C09062=1058.680,384.878,-115.207,174.460,37.992,157.227
C09063=1058.673,384.632,-115.166,174.454,37.986,157.226
C09064=1058.665,384.385,-115.126,174.449,37.979,157.224
C09065=1058.657,384.139,-115.086,174.443,37.972,157.222
C09066=1058.650,383.892,-115.045,174.437,37.965,157.221
C09067=1058.642,383.646,-115.004,174.432,37.959,157.219
C09068=1058.635,383.399,-114.964,174.427,37.952,157.217
C09069=1058.627,383.153,-114.923,174.420,37.945,157.215
C09070=1058.619,382.906,-114.883,174.415,37.939,157.214
C09071=1058.612,382.659,-114.842,174.409,37.932,157.212
C09072=1058.605,382.414,-114.802,174.404,37.926,157.210
C09073=1058.597,382.167,-114.762,174.399,37.919,157.209
C09074=1058.590,381.920,-114.720,174.392,37.912,157.207
C09075=1058.582,381.673,-114.681,174.387,37.906,157.205
C09076=1058.575,381.428,-114.640,174.382,37.899,157.204
C09077=1058.568,381.180,-114.600,174.377,37.893,157.202
C09078=1058.560,380.933,-114.560,174.371,37.886,157.200
C09079=1058.552,380.687,-114.519,174.366,37.880,157.199
C09080=1058.545,380.441,-114.479,174.360,37.873,157.197
C09081=1058.538,380.194,-114.439,174.354,37.867,157.195
C09082=1058.530,379.947,-114.399,174.349,37.860,157.194
C09083=1058.522,379.701,-114.359,174.344,37.854,157.192
C09084=1058.515,379.454,-114.319,174.339,37.848,157.191
C09085=1058.507,379.207,-114.279,174.333,37.841,157.189
C09086=1058.499,378.961,-114.239,174.327,37.835,157.187
C09087=1058.492,378.714,-114.200,174.322,37.829,157.186
C09088=1058.485,378.467,-114.160,174.317,37.822,157.184
C09089=1058.477,378.221,-114.120,174.311,37.816,157.183
C09090=1058.470,377.974,-114.080,174.306,37.810,157.181
C09091=1058.462,377.727,-114.040,174.301,37.803,157.179
C09092=1058.454,377.481,-114.000,174.296,37.797,157.178
C09093=1058.447,377.234,-113.961,174.291,37.791,157.176
C09094=1058.439,376.987,-113.921,174.285,37.785,157.175
C09095=1058.432,376.741,-113.881,174.280,37.778,157.173
C09096=1058.425,376.494,-113.841,174.274,37.772,157.172
C09097=1058.417,376.248,-113.802,174.269,37.766,157.170
C09098=1058.410,376.001,-113.762,174.264,37.760,157.168
C09099=1058.402,375.754,-113.723,174.258,37.753,157.167
C09100=1058.395,375.508,-113.683,174.253,37.747,157.165
C09101=1058.388,375.261,-113.644,174.248,37.741,157.164
C09102=1058.380,375.014,-113.604,174.243,37.735,157.162
C09103=1058.374,374.768,-113.565,174.238,37.729,157.161
C09104=1058.366,374.521,-113.525,174.232,37.723,157.159
C09105=1058.359,374.274,-113.485,174.227,37.717,157.158
C09106=1058.350,373.998,-113.441,174.222,37.709,157.156
C09107=1058.342,373.723,-113.397,174.216,37.703,157.154
C09108=1058.334,373.447,-113.353,174.210,37.696,157.152
C09109=1058.326,373.172,-113.309,174.204,37.689,157.151
C09110=1058.319,372.924,-113.270,174.199,37.683,157.149
C09111=1058.312,372.678,-113.231,174.194,37.677,157.148
C09112=1058.305,372.431,-113.192,174.189,37.671,157.146
C09113=1058.297,372.184,-113.152,174.184,37.665,157.145
C09114=1058.290,371.938,-113.114,174.179,37.659,157.143
C09115=1058.282,371.690,-113.074,174.174,37.653,157.142
C09116=1058.275,371.444,-113.035,174.169,37.647,157.140
C09117=1058.268,371.197,-112.997,174.164,37.641,157.139
C09118=1058.260,370.950,-112.957,174.159,37.635,157.137
C09119=1058.252,370.704,-112.918,174.154,37.630,157.136
C09120=1058.245,370.457,-112.880,174.149,37.624,157.134
C09121=1058.238,370.210,-112.840,174.144,37.618,157.133
C09122=1058.231,369.963,-112.802,174.139,37.612,157.131
C09123=1058.224,369.716,-112.763,174.134,37.606,157.130
C09124=1058.216,369.469,-112.723,174.128,37.600,157.129
C09125=1058.208,369.223,-112.685,174.123,37.594,157.127
C09126=1058.202,368.976,-112.646,174.118,37.588,157.126
C09127=1058.194,368.729,-112.607,174.113,37.582,157.124
C09128=1058.187,368.482,-112.569,174.109,37.577,157.123
C09129=1058.180,368.235,-112.530,174.104,37.571,157.121
C09130=1058.172,367.989,-112.492,174.099,37.565,157.120
C09131=1058.166,367.742,-112.453,174.094,37.559,157.119
C09132=1058.158,367.494,-112.414,174.089,37.554,157.117
C09133=1058.151,367.248,-112.375,174.084,37.548,157.116
C09134=1058.144,367.001,-112.337,174.079,37.542,157.114
C09135=1058.136,366.754,-112.298,174.075,37.536,157.113
C09136=1058.130,366.507,-112.260,174.070,37.531,157.112
C09137=1058.122,366.261,-112.222,174.065,37.525,157.110
C09138=1058.115,366.013,-112.183,174.060,37.519,157.109
C09139=1058.108,365.766,-112.144,174.055,37.514,157.107
C09140=1058.100,365.520,-112.106,174.051,37.508,157.106
C09141=1058.094,365.272,-112.068,174.046,37.502,157.105
C09142=1058.086,365.026,-112.029,174.041,37.497,157.103
C09143=1058.079,364.779,-111.991,174.036,37.491,157.102
C09144=1058.072,364.532,-111.952,174.031,37.485,157.100
C09145=1058.065,364.285,-111.914,174.027,37.480,157.099
C09146=1058.059,364.038,-111.875,174.022,37.474,157.098
C09147=1058.051,363.791,-111.838,174.017,37.469,157.096
C09148=1058.044,363.544,-111.800,174.012,37.462,157.095
C09149=1058.037,363.298,-111.761,174.007,37.457,157.093
C09150=1058.030,363.050,-111.723,174.003,37.451,157.092
C09151=1058.022,362.804,-111.685,173.998,37.446,157.091
C09152=1058.016,362.557,-111.647,173.993,37.440,157.089
C09153=1058.008,362.309,-111.609,173.988,37.435,157.088
C09154=1058.001,362.063,-111.571,173.984,37.429,157.087
C09155=1057.994,361.815,-111.533,173.979,37.424,157.085
C09156=1057.987,361.569,-111.495,173.974,37.419,157.084
C09157=1057.980,361.322,-111.457,173.969,37.413,157.083
C09158=1057.973,361.074,-111.419,173.965,37.408,157.081
C09159=1057.966,360.828,-111.381,173.960,37.402,157.080
C09160=1057.958,360.581,-111.343,173.955,37.397,157.079
C09161=1057.951,360.334,-111.306,173.951,37.391,157.077
C09162=1057.944,360.076,-111.266,173.946,37.386,157.076
C09163=1057.937,359.819,-111.227,173.941,37.380,157.075
C09164=1057.929,359.562,-111.187,173.936,37.375,157.073
C09165=1057.922,359.304,-111.148,173.931,37.369,157.072
C09166=1057.914,359.057,-111.111,173.926,37.364,157.071
C09167=1057.907,358.810,-111.073,173.922,37.358,157.069
C09168=1057.901,358.563,-111.035,173.917,37.353,157.068
C09169=1057.893,358.315,-110.997,173.912,37.347,157.067
C09170=1057.887,358.069,-110.960,173.908,37.342,157.066
C09171=1057.880,357.822,-110.923,173.904,37.337,157.064
C09172=1057.872,357.575,-110.885,173.899,37.331,157.063
C09173=1057.865,357.328,-110.848,173.895,37.326,157.062
C09174=1057.858,357.080,-110.810,173.890,37.321,157.060
C09175=1057.851,356.833,-110.773,173.886,37.316,157.059
C09176=1057.843,356.586,-110.735,173.881,37.310,157.058
C09177=1057.837,356.340,-110.698,173.876,37.305,157.057
C09178=1057.829,356.093,-110.660,173.872,37.300,157.055
C09179=1057.823,355.845,-110.622,173.867,37.295,157.054
C09180=1057.816,355.597,-110.585,173.862,37.289,157.053
C09181=1057.809,355.350,-110.548,173.859,37.284,157.052
C09182=1057.802,355.104,-110.511,173.854,37.279,157.050
C09183=1057.795,354.857,-110.473,173.850,37.274,157.049
C09184=1057.788,354.610,-110.436,173.845,37.269,157.048
C09185=1057.781,354.363,-110.399,173.840,37.264,157.047
C09186=1057.774,354.115,-110.362,173.836,37.258,157.045
C09187=1057.767,353.868,-110.324,173.831,37.253,157.044
C09188=1057.760,353.621,-110.287,173.827,37.248,157.043
C09189=1057.753,353.374,-110.250,173.823,37.243,157.042
C09190=1057.746,353.126,-110.213,173.818,37.238,157.040
C09191=1057.739,352.879,-110.176,173.814,37.232,157.039
C09192=1057.732,352.633,-110.139,173.809,37.227,157.038
C09193=1057.725,352.385,-110.102,173.805,37.222,157.037
C09194=1057.718,352.139,-110.065,173.800,37.217,157.035
C09195=1057.711,351.891,-110.029,173.796,37.212,157.034
C09196=1057.704,351.644,-109.991,173.792,37.207,157.033
C09197=1057.698,351.397,-109.955,173.788,37.202,157.032
C09198=1057.690,351.150,-109.917,173.783,37.197,157.031
C09199=1057.683,350.902,-109.880,173.779,37.192,157.029
C09200=1057.677,350.655,-109.844,173.774,37.187,157.028
C09201=1057.669,350.408,-109.807,173.770,37.182,157.027
C09202=1057.659,350.018,-109.749,173.763,37.174,157.025
C09203=1057.647,349.628,-109.691,173.756,37.166,157.023
C09204=1057.637,349.238,-109.633,173.750,37.158,157.021
C09205=1057.625,348.847,-109.576,173.742,37.151,157.020
C09206=1057.619,348.601,-109.539,173.739,37.145,157.018
C09207=1057.612,348.353,-109.502,173.734,37.140,157.017
C09208=1057.605,348.106,-109.466,173.730,37.135,157.016
C09209=1057.598,347.858,-109.429,173.726,37.130,157.015
C09210=1057.591,347.611,-109.393,173.721,37.125,157.014
C09211=1057.584,347.363,-109.356,173.717,37.120,157.012
C09212=1057.577,347.117,-109.320,173.713,37.116,157.011
C09213=1057.570,346.869,-109.283,173.709,37.111,157.010
C09214=1057.561,346.512,-109.230,173.703,37.103,157.008
C09215=1057.551,346.156,-109.178,173.697,37.097,157.007
C09216=1057.541,345.799,-109.125,173.690,37.089,157.005
C09217=1057.531,345.442,-109.074,173.684,37.083,157.004
C09218=1057.524,345.195,-109.037,173.680,37.078,157.002
C09219=1057.518,344.948,-109.000,173.676,37.073,157.001
C09220=1057.511,344.701,-108.965,173.672,37.068,157.000
C09221=1057.504,344.453,-108.928,173.667,37.063,156.999
C09222=1057.497,344.206,-108.892,173.663,37.058,156.998
C09223=1057.491,343.959,-108.856,173.659,37.054,156.997
C09224=1057.484,343.711,-108.819,173.655,37.049,156.996
C09225=1057.477,343.464,-108.783,173.651,37.044,156.994
C09226=1057.470,343.217,-108.747,173.646,37.039,156.993
C09227=1057.463,342.969,-108.712,173.643,37.035,156.992
C09228=1057.457,342.722,-108.675,173.639,37.029,156.991
C09229=1057.449,342.475,-108.639,173.634,37.025,156.990
C09230=1057.442,342.227,-108.604,173.630,37.020,156.989
C09231=1057.436,341.980,-108.567,173.626,37.015,156.988
C09232=1057.429,341.733,-108.531,173.622,37.011,156.987
C09233=1057.421,341.485,-108.496,173.618,37.006,156.986
C09234=1057.415,341.238,-108.460,173.614,37.001,156.984
C09235=1057.408,340.991,-108.424,173.610,36.997,156.983
C09236=1057.401,340.743,-108.388,173.606,36.992,156.982
C09237=1057.394,340.496,-108.352,173.601,36.987,156.981
C09238=1057.387,340.249,-108.317,173.598,36.983,156.980
C09239=1057.381,340.001,-108.281,173.594,36.978,156.979
C09240=1057.374,339.754,-108.245,173.589,36.973,156.978
C09241=1057.367,339.506,-108.209,173.586,36.969,156.977
C09242=1057.361,339.259,-108.173,173.582,36.964,156.976
C09243=1057.354,339.012,-108.138,173.577,36.959,156.975
C09244=1057.347,338.765,-108.103,173.573,36.955,156.974
C09245=1057.340,338.517,-108.066,173.570,36.950,156.972
C09246=1057.333,338.270,-108.031,173.565,36.945,156.971
C09247=1057.327,338.022,-107.996,173.561,36.941,156.970
C09248=1057.320,337.775,-107.959,173.557,36.936,156.969
C09249=1057.313,337.528,-107.924,173.554,36.932,156.968
C09250=1057.307,337.280,-107.889,173.549,36.927,156.967
C09251=1057.301,337.033,-107.853,173.545,36.922,156.966
C09252=1057.293,336.785,-107.817,173.542,36.917,156.965
C09253=1057.286,336.538,-107.782,173.537,36.913,156.964
C09254=1057.279,336.291,-107.747,173.533,36.908,156.963
C09255=1057.273,336.043,-107.712,173.530,36.904,156.962
C09256=1057.266,335.796,-107.676,173.526,36.899,156.961
C09257=1057.259,335.548,-107.641,173.521,36.895,156.960
C09258=1057.253,335.301,-107.606,173.518,36.890,156.959
C09259=1057.246,335.053,-107.570,173.514,36.886,156.958
C09260=1057.239,334.805,-107.535,173.510,36.881,156.956
C09261=1057.232,334.558,-107.500,173.506,36.877,156.955
C09262=1057.225,334.311,-107.465,173.502,36.872,156.954
C09263=1057.219,334.063,-107.430,173.498,36.868,156.953
C09264=1057.212,333.816,-107.394,173.494,36.863,156.952
C09265=1057.205,333.569,-107.359,173.490,36.859,156.951
C09266=1057.198,333.321,-107.324,173.486,36.854,156.950
C09267=1057.192,333.074,-107.289,173.482,36.850,156.949
C09268=1057.185,332.826,-107.254,173.479,36.846,156.948
C09269=1057.178,332.579,-107.219,173.475,36.841,156.947
C09270=1057.172,332.322,-107.182,173.470,36.836,156.946
C09271=1057.164,332.066,-107.146,173.467,36.831,156.945
C09272=1057.157,331.808,-107.109,173.463,36.827,156.944
C09273=1057.151,331.552,-107.073,173.458,36.822,156.943
C09274=1057.144,331.304,-107.038,173.455,36.818,156.942
C09275=1057.137,331.057,-107.003,173.451,36.813,156.941
C09276=1057.131,330.809,-106.968,173.447,36.809,156.940
C09277=1057.124,330.562,-106.933,173.444,36.805,156.939
C09278=1057.117,330.314,-106.898,173.440,36.800,156.938
C09279=1057.111,330.066,-106.864,173.436,36.796,156.937
C09280=1057.103,329.819,-106.829,173.432,36.792,156.936
C09281=1057.097,329.572,-106.794,173.428,36.787,156.935
C09282=1057.090,329.324,-106.760,173.425,36.783,156.934
C09283=1057.083,329.077,-106.725,173.421,36.779,156.933
C09284=1057.077,328.830,-106.691,173.416,36.774,156.932
C09285=1057.070,328.582,-106.656,173.413,36.770,156.931
C09286=1057.063,328.335,-106.622,173.409,36.766,156.930
C09287=1057.056,328.087,-106.587,173.406,36.762,156.929
C09288=1057.050,327.839,-106.552,173.402,36.757,156.928
C09289=1057.042,327.592,-106.518,173.398,36.753,156.927
C09290=1057.036,327.344,-106.483,173.395,36.749,156.926
C09291=1057.029,327.097,-106.448,173.390,36.744,156.925
C09292=1057.022,326.849,-106.414,173.386,36.740,156.924
C09293=1057.015,326.601,-106.380,173.383,36.735,156.923
C09294=1057.008,326.355,-106.346,173.379,36.732,156.922
C09295=1057.002,326.107,-106.311,173.376,36.727,156.921
C09296=1056.995,325.859,-106.277,173.372,36.723,156.920
C09297=1056.988,325.612,-106.243,173.368,36.719,156.919
C09298=1056.981,325.364,-106.208,173.365,36.714,156.918
C09299=1056.975,325.116,-106.174,173.360,36.710,156.917
C09300=1056.968,324.869,-106.140,173.357,36.706,156.916
C09301=1056.962,324.621,-106.105,173.353,36.702,156.915
C09302=1056.954,324.374,-106.071,173.349,36.697,156.914
C09303=1056.948,324.126,-106.037,173.346,36.693,156.913
C09304=1056.942,323.879,-106.002,173.342,36.689,156.912
C09305=1056.935,323.631,-105.968,173.339,36.685,156.911
C09306=1056.928,323.383,-105.934,173.335,36.681,156.911
C09307=1056.921,323.136,-105.900,173.331,36.676,156.910
C09308=1056.915,322.888,-105.866,173.328,36.672,156.909
C09309=1056.909,322.640,-105.832,173.324,36.668,156.908
C09310=1056.901,322.393,-105.798,173.321,36.664,156.907
C09311=1056.895,322.145,-105.763,173.317,36.660,156.906
C09312=1056.888,321.898,-105.729,173.313,36.655,156.905
C09313=1056.882,321.651,-105.695,173.310,36.651,156.904
C09314=1056.874,321.403,-105.661,173.306,36.647,156.903
C09315=1056.868,321.156,-105.627,173.302,36.643,156.902
C09316=1056.862,320.908,-105.592,173.298,36.639,156.901
C09317=1056.855,320.661,-105.559,173.295,36.635,156.900
C09318=1056.849,320.413,-105.525,173.291,36.630,156.899
C09319=1056.842,320.165,-105.491,173.287,36.626,156.898
C09320=1056.836,319.918,-105.457,173.284,36.622,156.897
C09321=1056.829,319.670,-105.423,173.280,36.618,156.896
C09322=1056.823,319.422,-105.389,173.277,36.613,156.895
C09323=1056.816,319.174,-105.356,173.273,36.609,156.894
C09324=1056.809,318.926,-105.321,173.270,36.605,156.893
C09325=1056.803,318.679,-105.288,173.266,36.601,156.892
C09326=1056.796,318.417,-105.252,173.262,36.597,156.892
C09327=1056.789,318.155,-105.216,173.259,36.592,156.891
C09328=1056.782,317.893,-105.180,173.255,36.588,156.890
C09329=1056.776,317.631,-105.145,173.252,36.584,156.889
C09330=1056.769,317.383,-105.110,173.248,36.579,156.888
C09331=1056.762,317.136,-105.077,173.244,36.575,156.887
C09332=1056.756,316.888,-105.043,173.241,36.571,156.886
C09333=1056.750,316.641,-105.010,173.237,36.567,156.885
C09334=1056.743,316.393,-104.975,173.234,36.563,156.884
C09335=1056.737,316.145,-104.942,173.230,36.558,156.883
C09336=1056.731,315.897,-104.908,173.227,36.554,156.882
C09337=1056.724,315.650,-104.875,173.223,36.550,156.881
C09338=1056.718,315.401,-104.841,173.220,36.546,156.880
C09339=1056.711,315.154,-104.807,173.216,36.542,156.879
C09340=1056.705,314.907,-104.773,173.213,36.538,156.878
C09341=1056.698,314.659,-104.740,173.210,36.534,156.877
C09342=1056.693,314.412,-104.706,173.206,36.530,156.877
C09343=1056.686,314.165,-104.673,173.203,36.526,156.876
C09344=1056.680,313.916,-104.639,173.199,36.522,156.875
C09345=1056.673,313.669,-104.606,173.196,36.518,156.874
C09346=1056.667,313.420,-104.572,173.192,36.513,156.873
C09347=1056.661,313.173,-104.539,173.189,36.510,156.872
C09348=1056.653,312.925,-104.506,173.185,36.506,156.871
C09349=1056.647,312.678,-104.473,173.182,36.502,156.870
C09350=1056.639,312.430,-104.439,173.178,36.498,156.869
C09351=1056.633,312.183,-104.407,173.174,36.493,156.868
C09352=1056.627,311.935,-104.374,173.171,36.489,156.868
C09353=1056.620,311.687,-104.340,173.168,36.485,156.867
C09354=1056.613,311.440,-104.307,173.165,36.482,156.866
C09355=1056.606,311.191,-104.274,173.161,36.478,156.865
C09356=1056.600,310.944,-104.241,173.158,36.474,156.864
C09357=1056.593,310.696,-104.208,173.154,36.470,156.863
C09358=1056.587,310.449,-104.175,173.151,36.466,156.862
C09359=1056.580,310.201,-104.142,173.147,36.462,156.861
C09360=1056.573,309.953,-104.109,173.144,36.458,156.861
C09361=1056.567,309.706,-104.076,173.140,36.454,156.860
C09362=1056.560,309.458,-104.043,173.137,36.450,156.859
C09363=1056.554,309.210,-104.010,173.134,36.446,156.858
C09364=1056.547,308.963,-103.978,173.131,36.442,156.857
C09365=1056.540,308.715,-103.945,173.127,36.439,156.856
C09366=1056.533,308.467,-103.912,173.124,36.435,156.855
C09367=1056.527,308.219,-103.879,173.120,36.431,156.854
C09368=1056.520,307.972,-103.845,173.117,36.427,156.854
C09369=1056.514,307.725,-103.813,173.113,36.423,156.853
C09370=1056.507,307.476,-103.780,173.111,36.419,156.852
C09371=1056.501,307.229,-103.747,173.107,36.415,156.851
C09372=1056.495,306.981,-103.714,173.104,36.411,156.850
C09373=1056.488,306.734,-103.682,173.100,36.407,156.849
C09374=1056.481,306.485,-103.649,173.097,36.404,156.848
C09375=1056.474,306.238,-103.616,173.093,36.400,156.848
C09376=1056.468,305.990,-103.583,173.091,36.396,156.847
C09377=1056.462,305.743,-103.551,173.087,36.391,156.846
C09378=1056.455,305.494,-103.518,173.084,36.388,156.845
C09379=1056.449,305.247,-103.485,173.080,36.384,156.844
C09380=1056.442,304.999,-103.452,173.077,36.380,156.843
C09381=1056.436,304.751,-103.421,173.073,36.376,156.843
C09382=1056.429,304.494,-103.386,173.071,36.372,156.842
C09383=1056.423,304.235,-103.352,173.067,36.368,156.841
C09384=1056.415,303.978,-103.318,173.064,36.364,156.840
C09385=1056.409,303.720,-103.285,173.060,36.360,156.839
C09386=1056.402,303.471,-103.252,173.057,36.356,156.838
C09387=1056.396,303.224,-103.219,173.053,36.352,156.837
C09388=1056.390,302.976,-103.186,173.050,36.348,156.836
C09389=1056.383,302.728,-103.155,173.047,36.345,156.836
C09390=1056.377,302.481,-103.122,173.044,36.341,156.835
C09391=1056.370,302.233,-103.089,173.040,36.337,156.834
C09392=1056.364,301.985,-103.056,173.037,36.333,156.833
C09393=1056.358,301.737,-103.024,173.034,36.329,156.832
C09394=1056.352,301.490,-102.992,173.031,36.325,156.831
C09395=1056.345,301.242,-102.960,173.027,36.321,156.830
C09396=1056.339,300.994,-102.928,173.024,36.317,156.830
C09397=1056.333,300.747,-102.895,173.021,36.313,156.829
C09398=1056.326,300.499,-102.862,173.018,36.310,156.828
C09399=1056.320,300.251,-102.830,173.014,36.306,156.827
C09400=1056.313,300.003,-102.798,173.011,36.302,156.826
C09401=1056.307,299.756,-102.765,173.009,36.298,156.825
C09402=1056.301,299.508,-102.733,173.005,36.294,156.824
C09403=1056.295,299.260,-102.700,173.002,36.290,156.824
C09404=1056.288,299.012,-102.669,172.999,36.287,156.823
C09405=1056.282,298.765,-102.636,172.996,36.283,156.822
C09406=1056.276,298.516,-102.604,172.992,36.279,156.821
C09407=1056.269,298.269,-102.571,172.989,36.275,156.820
C09408=1056.263,298.021,-102.539,172.986,36.271,156.819
C09409=1056.256,297.773,-102.507,172.983,36.267,156.819
C09410=1056.250,297.525,-102.475,172.979,36.263,156.818
C09411=1056.244,297.277,-102.442,172.977,36.259,156.817
C09412=1056.238,297.029,-102.410,172.973,36.256,156.816
C09413=1056.231,296.782,-102.378,172.970,36.252,156.815
C09414=1056.225,296.534,-102.346,172.967,36.248,156.814
C09415=1056.219,296.286,-102.314,172.964,36.244,156.814
C09416=1056.212,296.038,-102.283,172.960,36.240,156.813
C09417=1056.206,295.790,-102.250,172.958,36.237,156.812
C09418=1056.199,295.542,-102.219,172.955,36.233,156.811
C09419=1056.193,295.295,-102.188,172.951,36.229,156.810
C09420=1056.187,295.047,-102.155,172.949,36.226,156.810
C09421=1056.180,294.799,-102.123,172.945,36.222,156.809
C09422=1056.174,294.551,-102.091,172.942,36.218,156.808
C09423=1056.167,294.303,-102.060,172.939,36.214,156.807
C09424=1056.161,294.055,-102.028,172.936,36.211,156.806
C09425=1056.154,293.808,-101.996,172.932,36.206,156.805
C09426=1056.148,293.560,-101.964,172.930,36.203,156.805
C09427=1056.142,293.312,-101.932,172.927,36.199,156.804
C09428=1056.135,293.064,-101.901,172.923,36.195,156.803
C09429=1056.128,292.816,-101.869,172.921,36.192,156.802
C09430=1056.122,292.568,-101.837,172.917,36.188,156.801
C09431=1056.116,292.321,-101.806,172.914,36.184,156.801
C09432=1056.109,292.073,-101.775,172.911,36.181,156.800
C09433=1056.103,291.824,-101.743,172.908,36.177,156.799
C09434=1056.097,291.579,-101.711,172.904,36.173,156.798
C09435=1056.090,291.334,-101.681,172.902,36.170,156.797
C09436=1056.084,291.089,-101.649,172.899,36.166,156.797
C09437=1056.078,290.844,-101.618,172.896,36.162,156.796
C09438=1056.072,290.600,-101.587,172.893,36.159,156.795
C09439=1056.065,290.354,-101.556,172.890,36.155,156.794
C09440=1056.059,290.109,-101.524,172.887,36.151,156.793
C09441=1056.053,289.864,-101.493,172.883,36.148,156.793
C09442=1056.046,289.616,-101.462,172.881,36.144,156.792
C09443=1056.039,289.368,-101.430,172.878,36.140,156.791
C09444=1056.033,289.120,-101.398,172.875,36.136,156.790
C09445=1056.027,288.872,-101.367,172.872,36.133,156.790
C09446=1056.021,288.624,-101.337,172.868,36.129,156.789
C09447=1056.014,288.376,-101.305,172.866,36.125,156.788
C09448=1056.008,288.128,-101.273,172.862,36.122,156.787
C09449=1056.002,287.880,-101.242,172.860,36.118,156.786
C09450=1055.995,287.633,-101.211,172.857,36.114,156.786
C09451=1055.989,287.385,-101.180,172.853,36.111,156.785
C09452=1055.982,287.137,-101.149,172.851,36.107,156.784
C09453=1055.976,286.889,-101.117,172.847,36.104,156.783
C09454=1055.969,286.640,-101.086,172.845,36.100,156.782
C09455=1055.963,286.393,-101.055,172.842,36.096,156.782
C09456=1055.956,286.145,-101.024,172.839,36.093,156.781
C09457=1055.950,285.897,-100.993,172.836,36.089,156.780
C09458=1055.943,285.649,-100.962,172.832,36.085,156.779
C09459=1055.937,285.402,-100.931,172.830,36.081,156.778
C09460=1055.931,285.153,-100.900,172.826,36.078,156.778
C09461=1055.924,284.905,-100.869,172.824,36.074,156.777
C09462=1055.918,284.658,-100.837,172.821,36.070,156.776
C09463=1055.911,284.409,-100.807,172.818,36.067,156.775
C09464=1055.905,284.162,-100.775,172.815,36.063,156.775
C09465=1055.899,283.914,-100.745,172.812,36.060,156.774
C09466=1055.892,283.666,-100.714,172.809,36.056,156.773
C09467=1055.886,283.417,-100.683,172.807,36.052,156.772
C09468=1055.879,283.170,-100.652,172.803,36.049,156.771
C09469=1055.873,282.922,-100.621,172.801,36.045,156.771
C09470=1055.866,282.674,-100.590,172.797,36.042,156.770
C09471=1055.861,282.426,-100.559,172.795,36.038,156.769
C09472=1055.854,282.178,-100.528,172.792,36.034,156.768
C09473=1055.847,281.929,-100.497,172.789,36.031,156.768
C09474=1055.841,281.682,-100.466,172.786,36.027,156.767
C09475=1055.835,281.434,-100.435,172.783,36.023,156.766
C09476=1055.829,281.186,-100.405,172.780,36.019,156.765
C09477=1055.822,280.938,-100.374,172.777,36.016,156.764
C09478=1055.816,280.689,-100.343,172.774,36.012,156.764
C09479=1055.810,280.442,-100.312,172.772,36.009,156.763
C09480=1055.803,280.194,-100.281,172.768,36.005,156.762
C09481=1055.798,279.946,-100.251,172.766,36.001,156.761
C09482=1055.791,279.697,-100.220,172.762,35.998,156.761
C09483=1055.784,279.449,-100.189,172.760,35.994,156.760
C09484=1055.779,279.202,-100.158,172.757,35.991,156.759
C09485=1055.772,278.953,-100.127,172.754,35.987,156.758
C09486=1055.766,278.706,-100.098,172.751,35.984,156.758
C09487=1055.759,278.458,-100.066,172.749,35.980,156.757
C09488=1055.753,278.210,-100.036,172.745,35.976,156.756
C09489=1055.747,277.961,-100.005,172.743,35.972,156.755
C09490=1055.740,277.722,-99.976,172.739,35.969,156.755
C09491=1055.734,277.482,-99.947,172.737,35.966,156.754
C09492=1055.728,277.243,-99.917,172.735,35.962,156.753
C09493=1055.722,277.003,-99.888,172.731,35.959,156.752
C09494=1055.716,276.763,-99.858,172.729,35.955,156.752
C09495=1055.710,276.524,-99.828,172.726,35.952,156.751
C09496=1055.703,276.284,-99.800,172.723,35.948,156.750
C09497=1055.698,276.045,-99.770,172.721,35.945,156.749
C09498=1055.691,275.796,-99.739,172.717,35.941,156.749
C09499=1055.685,275.549,-99.709,172.715,35.938,156.748
C09500=1055.678,275.300,-99.678,172.713,35.934,156.747
C09501=1055.672,275.052,-99.648,172.709,35.931,156.746
C09502=1055.665,274.804,-99.618,172.707,35.927,156.746
C09503=1055.659,274.556,-99.588,172.703,35.924,156.745
C09504=1055.654,274.308,-99.557,172.701,35.920,156.744
C09505=1055.646,274.060,-99.527,172.699,35.916,156.743
C09506=1055.641,273.812,-99.497,172.695,35.912,156.743
C09507=1055.634,273.564,-99.466,172.693,35.909,156.742
C09508=1055.628,273.316,-99.436,172.689,35.905,156.741
C09509=1055.621,273.068,-99.406,172.687,35.902,156.740
C09510=1055.616,272.819,-99.376,172.685,35.898,156.740
C09511=1055.608,272.571,-99.346,172.681,35.895,156.739
C09512=1055.603,272.323,-99.315,172.679,35.891,156.738
C09513=1055.596,272.076,-99.286,172.676,35.888,156.737
C09514=1055.590,271.827,-99.255,172.673,35.884,156.737
C09515=1055.583,271.580,-99.225,172.671,35.881,156.736
C09516=1055.577,271.331,-99.195,172.667,35.877,156.735
C09517=1055.570,271.083,-99.166,172.665,35.873,156.734
C09518=1055.564,270.835,-99.135,172.662,35.870,156.734
C09519=1055.557,270.587,-99.105,172.659,35.866,156.733
C09520=1055.552,270.339,-99.075,172.657,35.863,156.732
C09521=1055.545,270.090,-99.045,172.654,35.859,156.731
C09522=1055.539,269.843,-99.015,172.651,35.856,156.731
C09523=1055.533,269.595,-98.986,172.649,35.852,156.730
C09524=1055.526,269.346,-98.955,172.646,35.849,156.729
C09525=1055.520,269.099,-98.925,172.643,35.845,156.728
C09526=1055.514,268.849,-98.895,172.640,35.842,156.728
C09527=1055.507,268.602,-98.866,172.637,35.838,156.727
C09528=1055.501,268.354,-98.835,172.635,35.834,156.726
C09529=1055.494,268.105,-98.806,172.632,35.831,156.725
C09530=1055.488,267.858,-98.776,172.629,35.827,156.725
C09531=1055.482,267.609,-98.747,172.627,35.824,156.724
C09532=1055.475,267.361,-98.716,172.624,35.820,156.723
C09533=1055.469,267.113,-98.686,172.621,35.817,156.723
C09534=1055.463,266.865,-98.657,172.619,35.813,156.722
C09535=1055.456,266.617,-98.627,172.616,35.810,156.721
C09536=1055.450,266.368,-98.597,172.613,35.806,156.720
C09537=1055.444,266.121,-98.567,172.611,35.803,156.720
C09538=1055.437,265.872,-98.538,172.607,35.799,156.719
C09539=1055.431,265.624,-98.508,172.605,35.795,156.718
C09540=1055.425,265.376,-98.479,172.603,35.792,156.717
C09541=1055.419,265.128,-98.450,172.599,35.788,156.717
C09542=1055.412,264.879,-98.419,172.597,35.785,156.716
C09543=1055.406,264.631,-98.390,172.595,35.781,156.715
C09544=1055.400,264.384,-98.360,172.592,35.778,156.714
C09545=1055.394,264.135,-98.330,172.589,35.774,156.714
C09546=1055.387,263.897,-98.302,172.587,35.771,156.713
C09547=1055.381,263.660,-98.274,172.584,35.767,156.712
C09548=1055.375,263.422,-98.245,172.582,35.764,156.712
C09549=1055.369,263.185,-98.217,172.580,35.761,156.711
C09550=1055.364,262.947,-98.189,172.576,35.757,156.710
C09551=1055.357,262.710,-98.161,172.574,35.754,156.709
C09552=1055.351,262.472,-98.133,172.572,35.750,156.709
C09553=1055.345,262.235,-98.105,172.569,35.748,156.708
C09554=1055.338,261.986,-98.075,172.566,35.744,156.707
C09555=1055.332,261.738,-98.046,172.564,35.740,156.707
C09556=1055.325,261.490,-98.017,172.561,35.737,156.706
C09557=1055.319,261.242,-97.988,172.559,35.733,156.705
C09558=1055.312,260.993,-97.958,172.555,35.730,156.704
C09559=1055.306,260.745,-97.929,172.553,35.727,156.704
C09560=1055.300,260.497,-97.900,172.551,35.723,156.703
C09561=1055.293,260.249,-97.871,172.547,35.720,156.702
C09562=1055.286,260.000,-97.842,172.545,35.716,156.702
C09563=1055.280,259.752,-97.813,172.543,35.713,156.701
C09564=1055.274,259.504,-97.784,172.540,35.709,156.700
C09565=1055.268,259.256,-97.754,172.537,35.705,156.699
C09566=1055.260,259.007,-97.726,172.535,35.702,156.699
C09567=1055.254,258.760,-97.696,172.532,35.699,156.698
C09568=1055.247,258.512,-97.667,172.530,35.695,156.697
C09569=1055.241,258.263,-97.638,172.527,35.692,156.697
C09570=1055.235,258.015,-97.609,172.524,35.688,156.696
C09571=1055.228,257.766,-97.579,172.522,35.685,156.695
C09572=1055.222,257.518,-97.550,172.520,35.681,156.694
C09573=1055.215,257.270,-97.521,172.516,35.678,156.694
C09574=1055.209,257.022,-97.492,172.514,35.674,156.693
C09575=1055.203,256.773,-97.464,172.512,35.671,156.692
C09576=1055.197,256.525,-97.435,172.509,35.667,156.691
C09577=1055.191,256.277,-97.406,172.507,35.664,156.691
C09578=1055.185,256.029,-97.377,172.504,35.660,156.690
C09579=1055.178,255.780,-97.347,172.501,35.657,156.689
C09580=1055.171,255.532,-97.318,172.499,35.653,156.689
C09581=1055.164,255.284,-97.290,172.497,35.650,156.688
C09582=1055.158,255.036,-97.261,172.494,35.647,156.687
C09583=1055.152,254.788,-97.232,172.491,35.643,156.686
C09584=1055.146,254.540,-97.203,172.489,35.639,156.686
C09585=1055.140,254.291,-97.174,172.486,35.636,156.685
C09586=1055.134,254.043,-97.145,172.484,35.632,156.684
C09587=1055.127,253.795,-97.116,172.482,35.629,156.684
C09588=1055.121,253.547,-97.087,172.478,35.625,156.683
C09589=1055.115,253.298,-97.058,172.476,35.622,156.682
C09590=1055.109,253.050,-97.030,172.474,35.618,156.681
C09591=1055.102,252.802,-97.002,172.471,35.614,156.681
C09592=1055.096,252.554,-96.973,172.469,35.611,156.680
C09593=1055.089,252.306,-96.943,172.467,35.608,156.679
C09594=1055.083,252.057,-96.915,172.463,35.604,156.679
C09595=1055.077,251.809,-96.886,172.461,35.601,156.678
C09596=1055.071,251.561,-96.857,172.459,35.597,156.677
C09597=1055.065,251.312,-96.829,172.456,35.594,156.676
C09598=1055.059,251.064,-96.800,172.454,35.590,156.676
C09599=1055.052,250.816,-96.771,172.452,35.586,156.675
C09600=1055.046,250.567,-96.743,172.449,35.583,156.674
C09601=1055.040,250.319,-96.714,172.446,35.579,156.673
C09602=1055.033,250.080,-96.686,172.444,35.576,156.673
C09603=1055.028,249.842,-96.658,172.441,35.573,156.672
C09604=1055.021,249.603,-96.631,172.439,35.569,156.671
C09605=1055.016,249.365,-96.604,172.437,35.566,156.671
C09606=1055.010,249.125,-96.576,172.434,35.562,156.670
C09607=1055.004,248.887,-96.548,172.432,35.559,156.669
C09608=1054.998,248.649,-96.521,172.430,35.555,156.668
C09609=1054.991,248.411,-96.494,172.428,35.552,156.668
C09610=1054.985,248.162,-96.465,172.425,35.548,156.667
C09611=1054.979,247.914,-96.436,172.423,35.545,156.666
C09612=1054.973,247.665,-96.408,172.421,35.541,156.666
C09613=1054.968,247.418,-96.379,172.418,35.538,156.665
C09614=1054.962,247.169,-96.351,172.416,35.534,156.664
C09615=1054.955,246.921,-96.322,172.414,35.530,156.663
C09616=1054.949,246.672,-96.294,172.410,35.527,156.663
C09617=1054.943,246.423,-96.266,172.408,35.523,156.662
C09618=1054.936,246.175,-96.237,172.406,35.520,156.661
C09619=1054.930,245.927,-96.209,172.403,35.516,156.660
C09620=1054.924,245.679,-96.180,172.401,35.513,156.660
C09621=1054.918,245.431,-96.152,172.399,35.510,156.659
C09622=1054.911,245.182,-96.124,172.396,35.506,156.658
C09623=1054.905,244.934,-96.095,172.394,35.502,156.658
C09624=1054.899,244.686,-96.067,172.392,35.499,156.657
C09625=1054.893,244.437,-96.039,172.389,35.495,156.656
C09626=1054.886,244.189,-96.010,172.387,35.492,156.655
C09627=1054.880,243.940,-95.982,172.385,35.488,156.655
C09628=1054.874,243.692,-95.954,172.381,35.484,156.654
C09629=1054.868,243.444,-95.927,172.379,35.481,156.653
C09630=1054.861,243.196,-95.898,172.377,35.477,156.653
C09631=1054.855,242.947,-95.869,172.375,35.474,156.652
C09632=1054.849,242.699,-95.842,172.372,35.470,156.651
C09633=1054.843,242.450,-95.813,172.370,35.467,156.650
C09634=1054.836,242.203,-95.785,172.368,35.464,156.650
C09635=1054.831,241.954,-95.757,172.365,35.460,156.649
C09636=1054.824,241.705,-95.729,172.363,35.456,156.648
C09637=1054.818,241.457,-95.701,172.361,35.453,156.648
C09638=1054.811,241.208,-95.673,172.358,35.449,156.647
C09639=1054.805,240.960,-95.645,172.356,35.446,156.646
C09640=1054.799,240.712,-95.617,172.354,35.442,156.645
C09641=1054.792,240.464,-95.589,172.351,35.439,156.645
C09642=1054.786,240.216,-95.561,172.349,35.435,156.644
C09643=1054.780,239.967,-95.533,172.347,35.432,156.643
C09644=1054.773,239.718,-95.505,172.345,35.428,156.643
C09645=1054.766,239.470,-95.477,172.342,35.425,156.642
C09646=1054.761,239.222,-95.449,172.340,35.421,156.641
C09647=1054.754,238.973,-95.422,172.338,35.418,156.640
C09648=1054.748,238.725,-95.394,172.335,35.414,156.640
C09649=1054.742,238.476,-95.366,172.333,35.411,156.639
C09650=1054.735,238.228,-95.338,172.331,35.407,156.638
C09651=1054.729,237.980,-95.311,172.328,35.404,156.638
C09652=1054.723,237.731,-95.282,172.326,35.400,156.637
C09653=1054.716,237.483,-95.255,172.324,35.397,156.636
C09654=1054.710,237.235,-95.227,172.321,35.393,156.635
C09655=1054.703,236.987,-95.199,172.319,35.389,156.635
C09656=1054.698,236.737,-95.172,172.317,35.386,156.634
C09657=1054.691,236.489,-95.144,172.315,35.383,156.633
C09658=1054.685,236.248,-95.117,172.312,35.379,156.633
C09659=1054.678,236.006,-95.090,172.310,35.376,156.632
C09660=1054.673,235.765,-95.063,172.308,35.372,156.631
C09661=1054.666,235.523,-95.036,172.305,35.369,156.631
C09662=1054.661,235.281,-95.009,172.303,35.365,156.630
C09663=1054.655,235.040,-94.982,172.301,35.362,156.629
C09664=1054.648,234.798,-94.956,172.299,35.358,156.628
C09665=1054.642,234.557,-94.929,172.296,35.355,156.628
C09666=1054.636,234.308,-94.902,172.294,35.352,156.627
C09667=1054.630,234.059,-94.873,172.292,35.348,156.626
C09668=1054.624,233.812,-94.846,172.289,35.344,156.626
C09669=1054.617,233.563,-94.818,172.287,35.341,156.625
C09670=1054.611,233.315,-94.791,172.285,35.337,156.624
C09671=1054.605,233.066,-94.764,172.282,35.334,156.623
C09672=1054.599,232.818,-94.736,172.280,35.330,156.623
C09673=1054.592,232.569,-94.708,172.278,35.326,156.622
C09674=1054.586,232.321,-94.681,172.277,35.323,156.621
C09675=1054.580,232.072,-94.653,172.274,35.319,156.621
C09676=1054.573,231.824,-94.626,172.272,35.316,156.620
C09677=1054.567,231.576,-94.599,172.270,35.312,156.619
C09678=1054.561,231.327,-94.571,172.267,35.308,156.618
C09679=1054.555,231.079,-94.544,172.265,35.305,156.618
C09680=1054.549,230.830,-94.516,172.263,35.302,156.617
C09681=1054.542,230.582,-94.489,172.261,35.298,156.616
C09682=1054.536,230.334,-94.461,172.258,35.295,156.616
C09683=1054.530,230.085,-94.434,172.256,35.291,156.615
C09684=1054.524,229.837,-94.407,172.254,35.287,156.614
C09685=1054.517,229.588,-94.380,172.251,35.284,156.613
C09686=1054.511,229.340,-94.352,172.249,35.280,156.613
C09687=1054.505,229.091,-94.326,172.247,35.277,156.612
C09688=1054.498,228.843,-94.298,172.246,35.273,156.611
C09689=1054.492,228.594,-94.271,172.243,35.269,156.611
C09690=1054.486,228.346,-94.243,172.241,35.266,156.610
C09691=1054.479,228.097,-94.216,172.239,35.263,156.609
C09692=1054.473,227.850,-94.190,172.236,35.259,156.608
C09693=1054.466,227.600,-94.163,172.234,35.256,156.608
C09694=1054.460,227.353,-94.135,172.232,35.252,156.607
C09695=1054.454,227.104,-94.108,172.230,35.248,156.606
C09696=1054.447,226.855,-94.081,172.227,35.245,156.606
C09697=1054.441,226.607,-94.054,172.225,35.241,156.605
C09698=1054.435,226.358,-94.027,172.223,35.238,156.604
C09699=1054.429,226.110,-93.999,172.221,35.234,156.603
C09700=1054.422,225.861,-93.973,172.219,35.230,156.603
C09701=1054.416,225.613,-93.946,172.217,35.227,156.602
C09702=1054.409,225.364,-93.919,172.215,35.224,156.601
C09703=1054.403,225.116,-93.892,172.212,35.220,156.601
C09704=1054.397,224.867,-93.865,172.210,35.217,156.600
C09705=1054.391,224.619,-93.838,172.208,35.213,156.599
C09706=1054.385,224.370,-93.811,172.205,35.209,156.599
C09707=1054.378,224.122,-93.785,172.204,35.206,156.598
C09708=1054.372,223.873,-93.758,172.202,35.202,156.597
C09709=1054.366,223.625,-93.730,172.200,35.199,156.596
C09710=1054.359,223.376,-93.703,172.197,35.195,156.596
C09711=1054.354,223.128,-93.677,172.195,35.191,156.595
C09712=1054.347,222.879,-93.650,172.193,35.188,156.594
C09713=1054.340,222.632,-93.623,172.190,35.184,156.593
C09714=1054.334,222.386,-93.596,172.189,35.181,156.593
C09715=1054.328,222.139,-93.570,172.187,35.177,156.592
C09716=1054.322,221.894,-93.543,172.185,35.173,156.591
C09717=1054.316,221.649,-93.517,172.182,35.170,156.591
C09718=1054.310,221.404,-93.490,172.180,35.166,156.590
C09719=1054.304,221.158,-93.463,172.179,35.162,156.589
C09720=1054.297,220.913,-93.437,172.177,35.159,156.589
C09721=1054.291,220.667,-93.411,172.174,35.156,156.588
C09722=1054.285,220.418,-93.384,172.172,35.152,156.587
C09723=1054.278,220.171,-93.357,172.170,35.149,156.586
C09724=1054.272,219.922,-93.331,172.168,35.145,156.586
C09725=1054.265,219.674,-93.304,172.166,35.141,156.585
C09726=1054.260,219.425,-93.278,172.164,35.138,156.584
C09727=1054.252,219.177,-93.251,172.162,35.134,156.583
C09728=1054.247,218.928,-93.224,172.159,35.131,156.583
C09729=1054.240,218.679,-93.197,172.157,35.127,156.582
C09730=1054.234,218.431,-93.171,172.156,35.123,156.581
C09731=1054.227,218.182,-93.144,172.154,35.120,156.581
C09732=1054.221,217.934,-93.118,172.151,35.116,156.580
C09733=1054.215,217.686,-93.092,172.149,35.112,156.579
C09734=1054.208,217.437,-93.065,172.147,35.109,156.578
C09735=1054.202,217.189,-93.039,172.145,35.105,156.578
C09736=1054.196,216.940,-93.012,172.143,35.102,156.577
C09737=1054.189,216.691,-92.986,172.141,35.098,156.576
C09738=1054.184,216.442,-92.960,172.139,35.094,156.576
C09739=1054.177,216.194,-92.933,172.136,35.091,156.575
C09740=1054.171,215.945,-92.907,172.135,35.087,156.574
C09741=1054.164,215.697,-92.880,172.133,35.084,156.573
C09742=1054.158,215.448,-92.853,172.131,35.080,156.573
C09743=1054.152,215.200,-92.827,172.128,35.076,156.572
C09744=1054.146,214.952,-92.801,172.127,35.073,156.571
C09745=1054.139,214.703,-92.774,172.125,35.069,156.571
C09746=1054.133,214.454,-92.748,172.123,35.065,156.570
C09747=1054.127,214.206,-92.722,172.120,35.062,156.569
C09748=1054.120,213.957,-92.695,172.119,35.058,156.568
C09749=1054.115,213.709,-92.669,172.117,35.055,156.568
C09750=1054.108,213.461,-92.643,172.114,35.051,156.567
C09751=1054.102,213.212,-92.616,172.112,35.047,156.566
C09752=1054.095,212.963,-92.590,172.111,35.044,156.566
C09753=1054.090,212.714,-92.564,172.109,35.040,156.565
C09754=1054.083,212.466,-92.538,172.106,35.037,156.564
C09755=1054.077,212.217,-92.511,172.104,35.033,156.563
C09756=1054.071,211.969,-92.485,172.103,35.029,156.563
C09757=1054.064,211.721,-92.459,172.101,35.026,156.562
C09758=1054.058,211.472,-92.433,172.098,35.022,156.561
C09759=1054.052,211.223,-92.407,172.096,35.018,156.561
C09760=1054.045,210.975,-92.381,172.095,35.015,156.560
C09761=1054.039,210.726,-92.354,172.093,35.011,156.559
C09762=1054.032,210.477,-92.328,172.090,35.007,156.558
C09763=1054.027,210.229,-92.302,172.088,35.003,156.558
C09764=1054.020,209.981,-92.276,172.087,35.000,156.557
C09765=1054.014,209.732,-92.250,172.085,34.996,156.556
C09766=1054.007,209.483,-92.224,172.082,34.993,156.555
C09767=1054.001,209.234,-92.198,172.081,34.989,156.555
C09768=1053.995,208.986,-92.172,172.079,34.985,156.554
C09769=1053.988,208.738,-92.146,172.077,34.982,156.553
C09770=1053.983,208.495,-92.120,172.074,34.978,156.553
C09771=1053.976,208.252,-92.095,172.073,34.974,156.552
C09772=1053.970,208.009,-92.069,172.071,34.971,156.551
C09773=1053.964,207.767,-92.045,172.068,34.967,156.550
C09774=1053.958,207.524,-92.019,172.067,34.964,156.550
C09775=1053.951,207.281,-91.994,172.065,34.961,156.549
C09776=1053.945,207.038,-91.969,172.063,34.957,156.548
C09777=1053.938,206.795,-91.943,172.062,34.953,156.548
C09778=1053.913,205.744,-91.838,171.850,34.861,156.532
C09779=1053.907,205.495,-91.813,171.848,34.858,156.532
C09780=1053.902,205.247,-91.788,171.845,34.855,156.531
C09781=1053.896,204.998,-91.764,171.843,34.852,156.531
C09782=1053.889,204.749,-91.738,171.840,34.849,156.530
C09783=1053.884,204.500,-91.714,171.838,34.846,156.530
C09784=1053.878,204.252,-91.689,171.836,34.843,156.529
C09785=1053.872,204.003,-91.664,171.833,34.841,156.529
C09786=1053.866,203.754,-91.639,171.830,34.838,156.528
C09787=1053.860,203.506,-91.614,171.828,34.835,156.528
C09788=1053.854,203.257,-91.590,171.826,34.832,156.527
C09789=1053.847,203.008,-91.564,171.823,34.829,156.526
C09790=1053.842,202.760,-91.540,171.821,34.827,156.526
C09791=1053.836,202.511,-91.515,171.819,34.824,156.525
C09792=1053.830,202.262,-91.490,171.816,34.821,156.525
C09793=1053.824,202.014,-91.465,171.813,34.818,156.524
C09794=1053.819,201.764,-91.440,171.811,34.815,156.524
C09795=1053.812,201.516,-91.417,171.809,34.812,156.523
C09796=1053.806,201.268,-91.391,171.807,34.810,156.523
C09797=1053.800,201.018,-91.367,171.804,34.807,156.522
C09798=1053.793,200.770,-91.342,171.801,34.804,156.522
C09799=1053.788,200.521,-91.318,171.799,34.802,156.521
C09800=1053.781,200.272,-91.294,171.797,34.799,156.521
C09801=1053.775,200.024,-91.268,171.794,34.796,156.520
C09802=1053.770,199.775,-91.244,171.792,34.794,156.520
C09803=1053.763,199.526,-91.220,171.790,34.791,156.519
C09804=1053.757,199.277,-91.195,171.787,34.788,156.519
C09805=1053.751,199.029,-91.171,171.784,34.785,156.518
C09806=1053.745,198.780,-91.147,171.782,34.783,156.518
C09807=1053.739,198.532,-91.123,171.780,34.780,156.517
C09808=1053.733,198.283,-91.098,171.778,34.777,156.517
C09809=1053.727,198.034,-91.073,171.775,34.774,156.516
C09810=1053.721,197.785,-91.049,171.772,34.772,156.516
C09811=1053.715,197.536,-91.025,171.770,34.769,156.515
C09812=1053.708,197.288,-91.000,171.768,34.766,156.515
C09813=1053.703,197.039,-90.976,171.765,34.764,156.514
C09814=1053.696,196.790,-90.952,171.763,34.761,156.514
C09815=1053.691,196.542,-90.927,171.761,34.758,156.513
C09816=1053.684,196.293,-90.903,171.759,34.756,156.513
C09817=1053.679,196.044,-90.879,171.756,34.753,156.512
C09818=1053.673,195.795,-90.854,171.753,34.750,156.512
C09819=1053.667,195.547,-90.830,171.751,34.748,156.511
C09820=1053.661,195.298,-90.805,171.749,34.745,156.511
C09821=1053.654,195.049,-90.781,171.747,34.742,156.510
C09822=1053.649,194.800,-90.757,171.745,34.740,156.510
C09823=1053.642,194.551,-90.733,171.741,34.736,156.509
C09824=1053.637,194.303,-90.709,171.739,34.734,156.509
C09825=1053.630,194.054,-90.685,171.737,34.732,156.508
C09826=1053.625,193.805,-90.661,171.735,34.729,156.508
C09827=1053.618,193.556,-90.637,171.733,34.726,156.507
C09828=1053.613,193.307,-90.612,171.731,34.723,156.507
C09829=1053.606,193.058,-90.588,171.728,34.721,156.506
C09830=1053.601,192.811,-90.563,171.725,34.718,156.506
C09831=1053.594,192.562,-90.539,171.723,34.715,156.505
C09832=1053.589,192.313,-90.515,171.721,34.713,156.505
C09833=1053.583,192.065,-90.491,171.719,34.710,156.504
C09834=1053.577,191.815,-90.468,171.717,34.707,156.504
C09835=1053.571,191.566,-90.444,171.714,34.705,156.503
C09836=1053.565,191.317,-90.419,171.712,34.702,156.503
C09837=1053.559,191.069,-90.396,171.709,34.699,156.502
C09838=1053.553,190.820,-90.371,171.707,34.697,156.502
C09839=1053.547,190.536,-90.343,171.704,34.693,156.501
C09840=1053.540,190.252,-90.316,171.702,34.690,156.501
C09841=1053.533,189.968,-90.288,171.700,34.687,156.500
C09842=1053.526,189.684,-90.261,171.697,34.684,156.500
C09843=1053.521,189.435,-90.237,171.694,34.682,156.499
C09844=1053.514,189.186,-90.213,171.692,34.679,156.499
C09845=1053.509,188.937,-90.189,171.690,34.677,156.498
C09846=1053.503,188.688,-90.165,171.688,34.674,156.498
C09847=1053.497,188.440,-90.142,171.685,34.671,156.497
C09848=1053.491,188.191,-90.117,171.683,34.669,156.497
C09849=1053.485,187.942,-90.093,171.681,34.666,156.496
C09850=1053.480,187.693,-90.069,171.678,34.663,156.496
C09851=1053.474,187.445,-90.046,171.676,34.660,156.495
C09852=1053.468,187.195,-90.022,171.674,34.658,156.495
C09853=1053.462,186.947,-89.998,171.672,34.655,156.494
C09854=1053.457,186.698,-89.974,171.670,34.652,156.494
C09855=1053.450,186.449,-89.950,171.668,34.650,156.493
C09856=1053.445,186.200,-89.926,171.665,34.647,156.493
C09857=1053.439,185.952,-89.902,171.662,34.645,156.492
C09858=1053.432,185.703,-89.878,171.660,34.642,156.492
C09859=1053.427,185.454,-89.855,171.658,34.639,156.491
C09860=1053.421,185.205,-89.831,171.656,34.637,156.491
C09861=1053.416,184.957,-89.807,171.654,34.634,156.490
C09862=1053.409,184.708,-89.783,171.652,34.631,156.490
C09863=1053.404,184.459,-89.759,171.650,34.629,156.489
C09864=1053.398,184.210,-89.736,171.647,34.626,156.489
C09865=1053.392,183.961,-89.712,171.645,34.624,156.488
C09866=1053.386,183.713,-89.689,171.643,34.621,156.488
C09867=1053.380,183.464,-89.665,171.640,34.619,156.487
C09868=1053.374,183.215,-89.642,171.638,34.616,156.487
C09869=1053.368,182.966,-89.618,171.636,34.614,156.487
C09870=1053.361,182.717,-89.595,171.634,34.611,156.486
C09871=1053.355,182.468,-89.571,171.632,34.609,156.486
C09872=1053.349,182.220,-89.548,171.629,34.606,156.485
C09873=1053.343,181.971,-89.524,171.627,34.604,156.485
C09874=1053.337,181.722,-89.501,171.625,34.601,156.484
C09875=1053.331,181.473,-89.479,171.623,34.599,156.484
C09876=1053.324,181.224,-89.455,171.621,34.596,156.483
C09877=1053.318,180.975,-89.432,171.618,34.594,156.483
C09878=1053.312,180.727,-89.408,171.616,34.592,156.483
C09879=1053.306,180.477,-89.385,171.614,34.589,156.482
C09880=1053.300,180.229,-89.361,171.611,34.587,156.482
C09881=1053.294,179.980,-89.338,171.609,34.584,156.481
C09882=1053.288,179.731,-89.315,171.607,34.582,156.481
C09883=1053.282,179.482,-89.291,171.605,34.579,156.480
C09884=1053.276,179.233,-89.268,171.603,34.577,156.480
C09885=1053.269,178.984,-89.244,171.601,34.574,156.479
C09886=1053.264,178.736,-89.221,171.599,34.572,156.479
C09887=1053.257,178.487,-89.199,171.597,34.569,156.478
C09888=1053.251,178.239,-89.175,171.594,34.567,156.478
C09889=1053.245,177.989,-89.152,171.592,34.564,156.478
C09890=1053.239,177.740,-89.129,171.589,34.561,156.477
C09891=1053.233,177.492,-89.105,171.587,34.559,156.477
C09892=1053.227,177.243,-89.083,171.585,34.556,156.476
C09893=1053.221,176.993,-89.059,171.583,34.555,156.476
C09894=1053.215,176.745,-89.036,171.581,34.552,156.475
C09895=1053.209,176.496,-89.013,171.579,34.550,156.475
C09896=1053.203,176.248,-88.990,171.576,34.547,156.475
C09897=1053.197,175.999,-88.967,171.574,34.545,156.474
C09898=1053.191,175.749,-88.944,171.572,34.542,156.474
C09899=1053.185,175.501,-88.920,171.570,34.540,156.473
C09900=1053.179,175.252,-88.897,171.568,34.537,156.473
C09901=1053.173,175.003,-88.874,171.566,34.534,156.472
C09902=1053.167,174.754,-88.851,171.564,34.532,156.472
C09903=1053.160,174.470,-88.825,171.562,34.529,156.471
C09904=1053.153,174.185,-88.798,171.558,34.526,156.471
C09905=1053.147,173.900,-88.773,171.556,34.524,156.470
C09906=1053.139,173.616,-88.746,171.554,34.521,156.470
C09907=1053.133,173.367,-88.723,171.552,34.518,156.469
C09908=1053.127,173.118,-88.700,171.550,34.516,156.469
C09909=1053.122,172.869,-88.677,171.548,34.514,156.468
C09910=1053.116,172.620,-88.654,171.546,34.511,156.468
C09911=1053.110,172.371,-88.631,171.544,34.509,156.468
C09912=1053.103,172.123,-88.608,171.542,34.506,156.467
C09913=1053.098,171.875,-88.585,171.539,34.504,156.467
C09914=1053.091,171.625,-88.562,171.537,34.501,156.466
C09915=1053.086,171.376,-88.539,171.535,34.499,156.466
C09916=1053.080,171.127,-88.516,171.533,34.496,156.465
C09917=1053.074,170.878,-88.493,171.531,34.494,156.465
C09918=1053.068,170.630,-88.471,171.529,34.491,156.464
C09919=1053.062,170.381,-88.448,171.527,34.489,156.464
C09920=1053.056,170.132,-88.425,171.525,34.487,156.464
C09921=1053.050,169.883,-88.402,171.522,34.484,156.463
C09922=1053.045,169.634,-88.379,171.520,34.482,156.463
C09923=1053.039,169.385,-88.356,171.518,34.479,156.462
C09924=1053.033,169.137,-88.334,171.516,34.477,156.462
C09925=1053.027,168.888,-88.311,171.514,34.474,156.461
C09926=1053.021,168.639,-88.288,171.512,34.472,156.461
C09927=1053.015,168.390,-88.265,171.510,34.469,156.460
C09928=1053.010,168.141,-88.242,171.508,34.467,156.460
C09929=1053.003,167.892,-88.220,171.506,34.464,156.460
C09930=1052.997,167.644,-88.197,171.503,34.462,156.459
C09931=1052.991,167.394,-88.173,171.501,34.460,156.459
C09932=1052.986,167.144,-88.151,171.499,34.457,156.458
C09933=1052.980,166.896,-88.128,171.497,34.455,156.458
C09934=1052.974,166.648,-88.106,171.495,34.452,156.457
C09935=1052.968,166.399,-88.083,171.493,34.450,156.457
C09936=1052.963,166.150,-88.060,171.491,34.447,156.456
C09937=1052.957,165.901,-88.037,171.490,34.445,156.456
C09938=1052.950,165.652,-88.015,171.488,34.442,156.456
C09939=1052.945,165.404,-87.992,171.485,34.440,156.455
C09940=1052.939,165.154,-87.970,171.483,34.438,156.455
C09941=1052.933,164.905,-87.947,171.481,34.435,156.454
C09942=1052.928,164.656,-87.924,171.479,34.433,156.454
C09943=1052.921,164.408,-87.902,171.477,34.430,156.453
C09944=1052.916,164.159,-87.879,171.475,34.428,156.453
C09945=1052.910,163.909,-87.856,171.473,34.425,156.452
C09946=1052.904,163.660,-87.833,171.471,34.422,156.452
C09947=1052.898,163.412,-87.811,171.469,34.420,156.452
C09948=1052.892,163.163,-87.788,171.466,34.417,156.451
C09949=1052.887,162.913,-87.766,171.464,34.415,156.451
C09950=1052.881,162.664,-87.743,171.463,34.412,156.450
C09951=1052.875,162.417,-87.721,171.461,34.411,156.450
C09952=1052.869,162.168,-87.698,171.459,34.408,156.449
C09953=1052.864,161.918,-87.676,171.457,34.405,156.449
C09954=1052.858,161.669,-87.653,171.455,34.403,156.449
C09955=1052.852,161.421,-87.630,171.453,34.400,156.448
C09956=1052.846,161.171,-87.608,171.451,34.398,156.448
C09957=1052.841,160.922,-87.585,171.448,34.395,156.447
C09958=1052.834,160.674,-87.563,171.446,34.393,156.447
C09959=1052.829,160.424,-87.541,171.444,34.391,156.446
C09960=1052.822,160.176,-87.518,171.443,34.388,156.446
C09961=1052.817,159.926,-87.496,171.441,34.386,156.445
C09962=1052.811,159.678,-87.474,171.439,34.384,156.445
C09963=1052.805,159.429,-87.453,171.437,34.381,156.445
C09964=1052.799,159.180,-87.430,171.435,34.379,156.444
C09965=1052.793,158.931,-87.408,171.433,34.376,156.444
C09966=1052.787,158.682,-87.385,171.431,34.374,156.443
C09967=1052.781,158.397,-87.360,171.428,34.372,156.443
C09968=1052.773,158.112,-87.334,171.426,34.369,156.442
C09969=1052.767,157.827,-87.309,171.424,34.366,156.442
C09970=1052.760,157.542,-87.283,171.421,34.364,156.442
C09971=1052.754,157.293,-87.262,171.419,34.361,156.441
C09972=1052.747,157.044,-87.239,171.418,34.359,156.441
C09973=1052.742,156.795,-87.217,171.416,34.357,156.440
C09974=1052.735,156.546,-87.195,171.414,34.354,156.440
C09975=1052.729,156.297,-87.173,171.412,34.352,156.439
C09976=1052.724,156.048,-87.151,171.410,34.350,156.439
C09977=1052.718,155.800,-87.129,171.407,34.347,156.439
C09978=1052.712,155.550,-87.107,171.405,34.345,156.438
C09979=1052.706,155.302,-87.084,171.403,34.343,156.438
C09980=1052.700,155.052,-87.063,171.401,34.340,156.437
C09981=1052.694,154.803,-87.041,171.400,34.338,156.437
C09982=1052.688,154.554,-87.018,171.398,34.335,156.436
C09983=1052.682,154.306,-86.997,171.396,34.333,156.436
C09984=1052.676,154.057,-86.975,171.394,34.331,156.436
C09985=1052.670,153.808,-86.953,171.392,34.329,156.435
C09986=1052.664,153.558,-86.931,171.390,34.326,156.435
C09987=1052.658,153.309,-86.909,171.387,34.324,156.434
C09988=1052.652,153.061,-86.887,171.385,34.322,156.434
C09989=1052.646,152.812,-86.865,171.384,34.319,156.434
C09990=1052.640,152.563,-86.844,171.382,34.317,156.433
C09991=1052.634,152.314,-86.821,171.380,34.315,156.433
C09992=1052.628,152.065,-86.799,171.378,34.312,156.432
C09993=1052.622,151.816,-86.778,171.376,34.310,156.432
C09994=1052.616,151.567,-86.756,171.374,34.308,156.432
C09995=1052.610,151.319,-86.734,171.372,34.305,156.431
C09996=1052.604,151.069,-86.712,171.371,34.303,156.431
//INST
///DATE 2021/06/17 10:56
///ATTR SC,RW,RJ
////FRAME ROBOT
///GROUP1 RB1
NOP
MOVL C00000 V=800.0 PL=0
MOVL C00001 V=800.0 PL=0
MOVL C00002 V=800.0 PL=0
MOVL C00003 V=800.0 PL=0
MOVL C00004 V=800.0 PL=0
MOVL C00005 V=800.0 PL=0
MOVL C00006 V=800.0 PL=0
MOVL C00007 V=800.0 PL=0
MOVL C00008 V=800.0 PL=0
MOVL C00009 V=800.0 PL=0
MOVL C00010 V=800.0 PL=0
MOVL C00011 V=800.0 PL=0
MOVL C00012 V=800.0 PL=0
MOVL C00013 V=800.0 PL=0
MOVL C00014 V=800.0 PL=0
MOVL C00015 V=800.0 PL=0
MOVL C00016 V=800.0 PL=0
MOVL C00017 V=800.0 PL=0
MOVL C00018 V=800.0 PL=0
MOVL C00019 V=800.0 PL=0
MOVL C00020 V=800.0 PL=0
MOVL C00021 V=800.0 PL=0
MOVL C00022 V=800.0 PL=0
MOVL C00023 V=800.0 PL=0
MOVL C00024 V=800.0 PL=0
MOVL C00025 V=800.0 PL=0
MOVL C00026 V=800.0 PL=0
MOVL C00027 V=800.0 PL=0
MOVL C00028 V=800.0 PL=0
MOVL C00029 V=800.0 PL=0
MOVL C00030 V=800.0 PL=0
MOVL C00031 V=800.0 PL=0
MOVL C00032 V=800.0 PL=0
MOVL C00033 V=800.0 PL=0
MOVL C00034 V=800.0 PL=0
MOVL C00035 V=800.0 PL=0
MOVL C00036 V=800.0 PL=0
MOVL C00037 V=800.0 PL=0
MOVL C00038 V=800.0 PL=0
MOVL C00039 V=800.0 PL=0
MOVL C00040 V=800.0 PL=0
MOVL C00041 V=800.0 PL=0
MOVL C00042 V=800.0 PL=0
MOVL C00043 V=800.0 PL=0
MOVL C00044 V=800.0 PL=0
MOVL C00045 V=800.0 PL=0
MOVL C00046 V=800.0 PL=0
MOVL C00047 V=800.0 PL=0
MOVL C00048 V=800.0 PL=0
MOVL C00049 V=800.0 PL=0
MOVL C00050 V=800.0 PL=0
MOVL C00051 V=800.0 PL=0
MOVL C00052 V=800.0 PL=0
MOVL C00053 V=800.0 PL=0
MOVL C00054 V=800.0 PL=0
MOVL C00055 V=800.0 PL=0
MOVL C00056 V=800.0 PL=0
MOVL C00057 V=800.0 PL=0
MOVL C00058 V=800.0 PL=0
MOVL C00059 V=800.0 PL=0
MOVL C00060 V=800.0 PL=0
MOVL C00061 V=800.0 PL=0
MOVL C00062 V=800.0 PL=0
MOVL C00063 V=800.0 PL=0
MOVL C00064 V=800.0 PL=0
MOVL C00065 V=800.0 PL=0
MOVL C00066 V=800.0 PL=0
MOVL C00067 V=800.0 PL=0
MOVL C00068 V=800.0 PL=0
MOVL C00069 V=800.0 PL=0
MOVL C00070 V=800.0 PL=0
MOVL C00071 V=800.0 PL=0
MOVL C00072 V=800.0 PL=0
MOVL C00073 V=800.0 PL=0
MOVL C00074 V=800.0 PL=0
MOVL C00075 V=800.0 PL=0
MOVL C00076 V=800.0 PL=0
MOVL C00077 V=800.0 PL=0
MOVL C00078 V=800.0 PL=0
MOVL C00079 V=800.0 PL=0
MOVL C00080 V=800.0 PL=0
MOVL C00081 V=800.0 PL=0
MOVL C00082 V=800.0 PL=0
MOVL C00083 V=800.0 PL=0
MOVL C00084 V=800.0 PL=0
MOVL C00085 V=800.0 PL=0
MOVL C00086 V=800.0 PL=0
MOVL C00087 V=800.0 PL=0
MOVL C00088 V=800.0 PL=0
MOVL C00089 V=800.0 PL=0
MOVL C00090 V=800.0 PL=0
MOVL C00091 V=800.0 PL=0
MOVL C00092 V=800.0 PL=0
MOVL C00093 V=800.0 PL=0
MOVL C00094 V=800.0 PL=0
MOVL C00095 V=800.0 PL=0
MOVL C00096 V=800.0 PL=0
MOVL C00097 V=800.0 PL=0
MOVL C00098 V=800.0 PL=0
MOVL C00099 V=800.0 PL=0
MOVL C00100 V=800.0 PL=0
MOVL C00101 V=800.0 PL=0
MOVL C00102 V=800.0 PL=0
MOVL C00103 V=800.0 PL=0
MOVL C00104 V=800.0 PL=0
MOVL C00105 V=800.0 PL=0
MOVL C00106 V=800.0 PL=0
MOVL C00107 V=800.0 PL=0
MOVL C00108 V=800.0 PL=0
MOVL C00109 V=800.0 PL=0
MOVL C00110 V=800.0 PL=0
MOVL C00111 V=800.0 PL=0
MOVL C00112 V=800.0 PL=0
MOVL C00113 V=800.0 PL=0
MOVL C00114 V=800.0 PL=0
MOVL C00115 V=800.0 PL=0
MOVL C00116 V=800.0 PL=0
MOVL C00117 V=800.0 PL=0
MOVL C00118 V=800.0 PL=0
MOVL C00119 V=800.0 PL=0
MOVL C00120 V=800.0 PL=0
MOVL C00121 V=800.0 PL=0
MOVL C00122 V=800.0 PL=0
MOVL C00123 V=800.0 PL=0
MOVL C00124 V=800.0 PL=0
MOVL C00125 V=800.0 PL=0
MOVL C00126 V=800.0 PL=0
MOVL C00127 V=800.0 PL=0
MOVL C00128 V=800.0 PL=0
MOVL C00129 V=800.0 PL=0
MOVL C00130 V=800.0 PL=0
MOVL C00131 V=800.0 PL=0
MOVL C00132 V=800.0 PL=0
MOVL C00133 V=800.0 PL=0
MOVL C00134 V=800.0 PL=0
MOVL C00135 V=800.0 PL=0
MOVL C00136 V=800.0 PL=0
MOVL C00137 V=800.0 PL=0
MOVL C00138 V=800.0 PL=0
MOVL C00139 V=800.0 PL=0
MOVL C00140 V=800.0 PL=0
MOVL C00141 V=800.0 PL=0
MOVL C00142 V=800.0 PL=0
MOVL C00143 V=800.0 PL=0
MOVL C00144 V=800.0 PL=0
MOVL C00145 V=800.0 PL=0
MOVL C00146 V=800.0 PL=0
MOVL C00147 V=800.0 PL=0
MOVL C00148 V=800.0 PL=0
MOVL C00149 V=800.0 PL=0
MOVL C00150 V=800.0 PL=0
MOVL C00151 V=800.0 PL=0
MOVL C00152 V=800.0 PL=0
MOVL C00153 V=800.0 PL=0
MOVL C00154 V=800.0 PL=0
MOVL C00155 V=800.0 PL=0
MOVL C00156 V=800.0 PL=0
MOVL C00157 V=800.0 PL=0
MOVL C00158 V=800.0 PL=0
MOVL C00159 V=800.0 PL=0
MOVL C00160 V=800.0 PL=0
MOVL C00161 V=800.0 PL=0
MOVL C00162 V=800.0 PL=0
MOVL C00163 V=800.0 PL=0
MOVL C00164 V=800.0 PL=0
MOVL C00165 V=800.0 PL=0
MOVL C00166 V=800.0 PL=0
MOVL C00167 V=800.0 PL=0
MOVL C00168 V=800.0 PL=0
MOVL C00169 V=800.0 PL=0
MOVL C00170 V=800.0 PL=0
MOVL C00171 V=800.0 PL=0
MOVL C00172 V=800.0 PL=0
MOVL C00173 V=800.0 PL=0
MOVL C00174 V=800.0 PL=0
MOVL C00175 V=800.0 PL=0
MOVL C00176 V=800.0 PL=0
MOVL C00177 V=800.0 PL=0
MOVL C00178 V=800.0 PL=0
MOVL C00179 V=800.0 PL=0
MOVL C00180 V=800.0 PL=0
MOVL C00181 V=800.0 PL=0
MOVL C00182 V=800.0 PL=0
MOVL C00183 V=800.0 PL=0
MOVL C00184 V=800.0 PL=0
MOVL C00185 V=800.0 PL=0
MOVL C00186 V=800.0 PL=0
MOVL C00187 V=800.0 PL=0
MOVL C00188 V=800.0 PL=0
MOVL C00189 V=800.0 PL=0
MOVL C00190 V=800.0 PL=0
MOVL C00191 V=800.0 PL=0
MOVL C00192 V=800.0 PL=0
MOVL C00193 V=800.0 PL=0
MOVL C00194 V=800.0 PL=0
MOVL C00195 V=800.0 PL=0
MOVL C00196 V=800.0 PL=0
MOVL C00197 V=800.0 PL=0
MOVL C00198 V=800.0 PL=0
MOVL C00199 V=800.0 PL=0
MOVL C00200 V=800.0 PL=0
MOVL C00201 V=800.0 PL=0
MOVL C00202 V=800.0 PL=0
MOVL C00203 V=800.0 PL=0
MOVL C00204 V=800.0 PL=0
MOVL C00205 V=800.0 PL=0
MOVL C00206 V=800.0 PL=0
MOVL C00207 V=800.0 PL=0
MOVL C00208 V=800.0 PL=0
MOVL C00209 V=800.0 PL=0
MOVL C00210 V=800.0 PL=0
MOVL C00211 V=800.0 PL=0
MOVL C00212 V=800.0 PL=0
MOVL C00213 V=800.0 PL=0
MOVL C00214 V=800.0 PL=0
MOVL C00215 V=800.0 PL=0
MOVL C00216 V=800.0 PL=0
MOVL C00217 V=800.0 PL=0
MOVL C00218 V=800.0 PL=0
MOVL C00219 V=800.0 PL=0
MOVL C00220 V=800.0 PL=0
MOVL C00221 V=800.0 PL=0
MOVL C00222 V=800.0 PL=0
MOVL C00223 V=800.0 PL=0
MOVL C00224 V=800.0 PL=0
MOVL C00225 V=800.0 PL=0
MOVL C00226 V=800.0 PL=0
MOVL C00227 V=800.0 PL=0
MOVL C00228 V=800.0 PL=0
MOVL C00229 V=800.0 PL=0
MOVL C00230 V=800.0 PL=0
MOVL C00231 V=800.0 PL=0
MOVL C00232 V=800.0 PL=0
MOVL C00233 V=800.0 PL=0
MOVL C00234 V=800.0 PL=0
MOVL C00235 V=800.0 PL=0
MOVL C00236 V=800.0 PL=0
MOVL C00237 V=800.0 PL=0
MOVL C00238 V=800.0 PL=0
MOVL C00239 V=800.0 PL=0
MOVL C00240 V=800.0 PL=0
MOVL C00241 V=800.0 PL=0
MOVL C00242 V=800.0 PL=0
MOVL C00243 V=800.0 PL=0
MOVL C00244 V=800.0 PL=0
MOVL C00245 V=800.0 PL=0
MOVL C00246 V=800.0 PL=0
MOVL C00247 V=800.0 PL=0
MOVL C00248 V=800.0 PL=0
MOVL C00249 V=800.0 PL=0
MOVL C00250 V=800.0 PL=0
MOVL C00251 V=800.0 PL=0
MOVL C00252 V=800.0 PL=0
MOVL C00253 V=800.0 PL=0
MOVL C00254 V=800.0 PL=0
MOVL C00255 V=800.0 PL=0
MOVL C00256 V=800.0 PL=0
MOVL C00257 V=800.0 PL=0
MOVL C00258 V=800.0 PL=0
MOVL C00259 V=800.0 PL=0
MOVL C00260 V=800.0 PL=0
MOVL C00261 V=800.0 PL=0
MOVL C00262 V=800.0 PL=0
MOVL C00263 V=800.0 PL=0
MOVL C00264 V=800.0 PL=0
MOVL C00265 V=800.0 PL=0
MOVL C00266 V=800.0 PL=0
MOVL C00267 V=800.0 PL=0
MOVL C00268 V=800.0 PL=0
MOVL C00269 V=800.0 PL=0
MOVL C00270 V=800.0 PL=0
MOVL C00271 V=800.0 PL=0
MOVL C00272 V=800.0 PL=0
MOVL C00273 V=800.0 PL=0
MOVL C00274 V=800.0 PL=0
MOVL C00275 V=800.0 PL=0
MOVL C00276 V=800.0 PL=0
MOVL C00277 V=800.0 PL=0
MOVL C00278 V=800.0 PL=0
MOVL C00279 V=800.0 PL=0
MOVL C00280 V=800.0 PL=0
MOVL C00281 V=800.0 PL=0
MOVL C00282 V=800.0 PL=0
MOVL C00283 V=800.0 PL=0
MOVL C00284 V=800.0 PL=0
MOVL C00285 V=800.0 PL=0
MOVL C00286 V=800.0 PL=0
MOVL C00287 V=800.0 PL=0
MOVL C00288 V=800.0 PL=0
MOVL C00289 V=800.0 PL=0
MOVL C00290 V=800.0 PL=0
MOVL C00291 V=800.0 PL=0
MOVL C00292 V=800.0 PL=0
MOVL C00293 V=800.0 PL=0
MOVL C00294 V=800.0 PL=0
MOVL C00295 V=800.0 PL=0
MOVL C00296 V=800.0 PL=0
MOVL C00297 V=800.0 PL=0
MOVL C00298 V=800.0 PL=0
MOVL C00299 V=800.0 PL=0
MOVL C00300 V=800.0 PL=0
MOVL C00301 V=800.0 PL=0
MOVL C00302 V=800.0 PL=0
MOVL C00303 V=800.0 PL=0
MOVL C00304 V=800.0 PL=0
MOVL C00305 V=800.0 PL=0
MOVL C00306 V=800.0 PL=0
MOVL C00307 V=800.0 PL=0
MOVL C00308 V=800.0 PL=0
MOVL C00309 V=800.0 PL=0
MOVL C00310 V=800.0 PL=0
MOVL C00311 V=800.0 PL=0
MOVL C00312 V=800.0 PL=0
MOVL C00313 V=800.0 PL=0
MOVL C00314 V=800.0 PL=0
MOVL C00315 V=800.0 PL=0
MOVL C00316 V=800.0 PL=0
MOVL C00317 V=800.0 PL=0
MOVL C00318 V=800.0 PL=0
MOVL C00319 V=800.0 PL=0
MOVL C00320 V=800.0 PL=0
MOVL C00321 V=800.0 PL=0
MOVL C00322 V=800.0 PL=0
MOVL C00323 V=800.0 PL=0
MOVL C00324 V=800.0 PL=0
MOVL C00325 V=800.0 PL=0
MOVL C00326 V=800.0 PL=0
MOVL C00327 V=800.0 PL=0
MOVL C00328 V=800.0 PL=0
MOVL C00329 V=800.0 PL=0
MOVL C00330 V=800.0 PL=0
MOVL C00331 V=800.0 PL=0
MOVL C00332 V=800.0 PL=0
MOVL C00333 V=800.0 PL=0
MOVL C00334 V=800.0 PL=0
MOVL C00335 V=800.0 PL=0
MOVL C00336 V=800.0 PL=0
MOVL C00337 V=800.0 PL=0
MOVL C00338 V=800.0 PL=0
MOVL C00339 V=800.0 PL=0
MOVL C00340 V=800.0 PL=0
MOVL C00341 V=800.0 PL=0
MOVL C00342 V=800.0 PL=0
MOVL C00343 V=800.0 PL=0
MOVL C00344 V=800.0 PL=0
MOVL C00345 V=800.0 PL=0
MOVL C00346 V=800.0 PL=0
MOVL C00347 V=800.0 PL=0
MOVL C00348 V=800.0 PL=0
MOVL C00349 V=800.0 PL=0
MOVL C00350 V=800.0 PL=0
MOVL C00351 V=800.0 PL=0
MOVL C00352 V=800.0 PL=0
MOVL C00353 V=800.0 PL=0
MOVL C00354 V=800.0 PL=0
MOVL C00355 V=800.0 PL=0
MOVL C00356 V=800.0 PL=0
MOVL C00357 V=800.0 PL=0
MOVL C00358 V=800.0 PL=0
MOVL C00359 V=800.0 PL=0
MOVL C00360 V=800.0 PL=0
MOVL C00361 V=800.0 PL=0
MOVL C00362 V=800.0 PL=0
MOVL C00363 V=800.0 PL=0
MOVL C00364 V=800.0 PL=0
MOVL C00365 V=800.0 PL=0
MOVL C00366 V=800.0 PL=0
MOVL C00367 V=800.0 PL=0
MOVL C00368 V=800.0 PL=0
MOVL C00369 V=800.0 PL=0
MOVL C00370 V=800.0 PL=0
MOVL C00371 V=800.0 PL=0
MOVL C00372 V=800.0 PL=0
MOVL C00373 V=800.0 PL=0
MOVL C00374 V=800.0 PL=0
MOVL C00375 V=800.0 PL=0
MOVL C00376 V=800.0 PL=0
MOVL C00377 V=800.0 PL=0
MOVL C00378 V=800.0 PL=0
MOVL C00379 V=800.0 PL=0
MOVL C00380 V=800.0 PL=0
MOVL C00381 V=800.0 PL=0
MOVL C00382 V=800.0 PL=0
MOVL C00383 V=800.0 PL=0
MOVL C00384 V=800.0 PL=0
MOVL C00385 V=800.0 PL=0
MOVL C00386 V=800.0 PL=0
MOVL C00387 V=800.0 PL=0
MOVL C00388 V=800.0 PL=0
MOVL C00389 V=800.0 PL=0
MOVL C00390 V=800.0 PL=0
MOVL C00391 V=800.0 PL=0
MOVL C00392 V=800.0 PL=0
MOVL C00393 V=800.0 PL=0
MOVL C00394 V=800.0 PL=0
MOVL C00395 V=800.0 PL=0
MOVL C00396 V=800.0 PL=0
MOVL C00397 V=800.0 PL=0
MOVL C00398 V=800.0 PL=0
MOVL C00399 V=800.0 PL=0
MOVL C00400 V=800.0 PL=0
MOVL C00401 V=800.0 PL=0
MOVL C00402 V=800.0 PL=0
MOVL C00403 V=800.0 PL=0
MOVL C00404 V=800.0 PL=0
MOVL C00405 V=800.0 PL=0
MOVL C00406 V=800.0 PL=0
MOVL C00407 V=800.0 PL=0
MOVL C00408 V=800.0 PL=0
MOVL C00409 V=800.0 PL=0
MOVL C00410 V=800.0 PL=0
MOVL C00411 V=800.0 PL=0
MOVL C00412 V=800.0 PL=0
MOVL C00413 V=800.0 PL=0
MOVL C00414 V=800.0 PL=0
MOVL C00415 V=800.0 PL=0
MOVL C00416 V=800.0 PL=0
MOVL C00417 V=800.0 PL=0
MOVL C00418 V=800.0 PL=0
MOVL C00419 V=800.0 PL=0
MOVL C00420 V=800.0 PL=0
MOVL C00421 V=800.0 PL=0
MOVL C00422 V=800.0 PL=0
MOVL C00423 V=800.0 PL=0
MOVL C00424 V=800.0 PL=0
MOVL C00425 V=800.0 PL=0
MOVL C00426 V=800.0 PL=0
MOVL C00427 V=800.0 PL=0
MOVL C00428 V=800.0 PL=0
MOVL C00429 V=800.0 PL=0
MOVL C00430 V=800.0 PL=0
MOVL C00431 V=800.0 PL=0
MOVL C00432 V=800.0 PL=0
MOVL C00433 V=800.0 PL=0
MOVL C00434 V=800.0 PL=0
MOVL C00435 V=800.0 PL=0
MOVL C00436 V=800.0 PL=0
MOVL C00437 V=800.0 PL=0
MOVL C00438 V=800.0 PL=0
MOVL C00439 V=800.0 PL=0
MOVL C00440 V=800.0 PL=0
MOVL C00441 V=800.0 PL=0
MOVL C00442 V=800.0 PL=0
MOVL C00443 V=800.0 PL=0
MOVL C00444 V=800.0 PL=0
MOVL C00445 V=800.0 PL=0
MOVL C00446 V=800.0 PL=0
MOVL C00447 V=800.0 PL=0
MOVL C00448 V=800.0 PL=0
MOVL C00449 V=800.0 PL=0
MOVL C00450 V=800.0 PL=0
MOVL C00451 V=800.0 PL=0
MOVL C00452 V=800.0 PL=0
MOVL C00453 V=800.0 PL=0
MOVL C00454 V=800.0 PL=0
MOVL C00455 V=800.0 PL=0
MOVL C00456 V=800.0 PL=0
MOVL C00457 V=800.0 PL=0
MOVL C00458 V=800.0 PL=0
MOVL C00459 V=800.0 PL=0
MOVL C00460 V=800.0 PL=0
MOVL C00461 V=800.0 PL=0
MOVL C00462 V=800.0 PL=0
MOVL C00463 V=800.0 PL=0
MOVL C00464 V=800.0 PL=0
MOVL C00465 V=800.0 PL=0
MOVL C00466 V=800.0 PL=0
MOVL C00467 V=800.0 PL=0
MOVL C00468 V=800.0 PL=0
MOVL C00469 V=800.0 PL=0
MOVL C00470 V=800.0 PL=0
MOVL C00471 V=800.0 PL=0
MOVL C00472 V=800.0 PL=0
MOVL C00473 V=800.0 PL=0
MOVL C00474 V=800.0 PL=0
MOVL C00475 V=800.0 PL=0
MOVL C00476 V=800.0 PL=0
MOVL C00477 V=800.0 PL=0
MOVL C00478 V=800.0 PL=0
MOVL C00479 V=800.0 PL=0
MOVL C00480 V=800.0 PL=0
MOVL C00481 V=800.0 PL=0
MOVL C00482 V=800.0 PL=0
MOVL C00483 V=800.0 PL=0
MOVL C00484 V=800.0 PL=0
MOVL C00485 V=800.0 PL=0
MOVL C00486 V=800.0 PL=0
MOVL C00487 V=800.0 PL=0
MOVL C00488 V=800.0 PL=0
MOVL C00489 V=800.0 PL=0
MOVL C00490 V=800.0 PL=0
MOVL C00491 V=800.0 PL=0
MOVL C00492 V=800.0 PL=0
MOVL C00493 V=800.0 PL=0
MOVL C00494 V=800.0 PL=0
MOVL C00495 V=800.0 PL=0
MOVL C00496 V=800.0 PL=0
MOVL C00497 V=800.0 PL=0
MOVL C00498 V=800.0 PL=0
MOVL C00499 V=800.0 PL=0
MOVL C00500 V=800.0 PL=0
MOVL C00501 V=800.0 PL=0
MOVL C00502 V=800.0 PL=0
MOVL C00503 V=800.0 PL=0
MOVL C00504 V=800.0 PL=0
MOVL C00505 V=800.0 PL=0
MOVL C00506 V=800.0 PL=0
MOVL C00507 V=800.0 PL=0
MOVL C00508 V=800.0 PL=0
MOVL C00509 V=800.0 PL=0
MOVL C00510 V=800.0 PL=0
MOVL C00511 V=800.0 PL=0
MOVL C00512 V=800.0 PL=0
MOVL C00513 V=800.0 PL=0
MOVL C00514 V=800.0 PL=0
MOVL C00515 V=800.0 PL=0
MOVL C00516 V=800.0 PL=0
MOVL C00517 V=800.0 PL=0
MOVL C00518 V=800.0 PL=0
MOVL C00519 V=800.0 PL=0
MOVL C00520 V=800.0 PL=0
MOVL C00521 V=800.0 PL=0
MOVL C00522 V=800.0 PL=0
MOVL C00523 V=800.0 PL=0
MOVL C00524 V=800.0 PL=0
MOVL C00525 V=800.0 PL=0
MOVL C00526 V=800.0 PL=0
MOVL C00527 V=800.0 PL=0
MOVL C00528 V=800.0 PL=0
MOVL C00529 V=800.0 PL=0
MOVL C00530 V=800.0 PL=0
MOVL C00531 V=800.0 PL=0
MOVL C00532 V=800.0 PL=0
MOVL C00533 V=800.0 PL=0
MOVL C00534 V=800.0 PL=0
MOVL C00535 V=800.0 PL=0
MOVL C00536 V=800.0 PL=0
MOVL C00537 V=800.0 PL=0
MOVL C00538 V=800.0 PL=0
MOVL C00539 V=800.0 PL=0
MOVL C00540 V=800.0 PL=0
MOVL C00541 V=800.0 PL=0
MOVL C00542 V=800.0 PL=0
MOVL C00543 V=800.0 PL=0
MOVL C00544 V=800.0 PL=0
MOVL C00545 V=800.0 PL=0
MOVL C00546 V=800.0 PL=0
MOVL C00547 V=800.0 PL=0
MOVL C00548 V=800.0 PL=0
MOVL C00549 V=800.0 PL=0
MOVL C00550 V=800.0 PL=0
MOVL C00551 V=800.0 PL=0
MOVL C00552 V=800.0 PL=0
MOVL C00553 V=800.0 PL=0
MOVL C00554 V=800.0 PL=0
MOVL C00555 V=800.0 PL=0
MOVL C00556 V=800.0 PL=0
MOVL C00557 V=800.0 PL=0
MOVL C00558 V=800.0 PL=0
MOVL C00559 V=800.0 PL=0
MOVL C00560 V=800.0 PL=0
MOVL C00561 V=800.0 PL=0
MOVL C00562 V=800.0 PL=0
MOVL C00563 V=800.0 PL=0
MOVL C00564 V=800.0 PL=0
MOVL C00565 V=800.0 PL=0
MOVL C00566 V=800.0 PL=0
MOVL C00567 V=800.0 PL=0
MOVL C00568 V=800.0 PL=0
MOVL C00569 V=800.0 PL=0
MOVL C00570 V=800.0 PL=0
MOVL C00571 V=800.0 PL=0
MOVL C00572 V=800.0 PL=0
MOVL C00573 V=800.0 PL=0
MOVL C00574 V=800.0 PL=0
MOVL C00575 V=800.0 PL=0
MOVL C00576 V=800.0 PL=0
MOVL C00577 V=800.0 PL=0
MOVL C00578 V=800.0 PL=0
MOVL C00579 V=800.0 PL=0
MOVL C00580 V=800.0 PL=0
MOVL C00581 V=800.0 PL=0
MOVL C00582 V=800.0 PL=0
MOVL C00583 V=800.0 PL=0
MOVL C00584 V=800.0 PL=0
MOVL C00585 V=800.0 PL=0
MOVL C00586 V=800.0 PL=0
MOVL C00587 V=800.0 PL=0
MOVL C00588 V=800.0 PL=0
MOVL C00589 V=800.0 PL=0
MOVL C00590 V=800.0 PL=0
MOVL C00591 V=800.0 PL=0
MOVL C00592 V=800.0 PL=0
MOVL C00593 V=800.0 PL=0
MOVL C00594 V=800.0 PL=0
MOVL C00595 V=800.0 PL=0
MOVL C00596 V=800.0 PL=0
MOVL C00597 V=800.0 PL=0
MOVL C00598 V=800.0 PL=0
MOVL C00599 V=800.0 PL=0
MOVL C00600 V=800.0 PL=0
MOVL C00601 V=800.0 PL=0
MOVL C00602 V=800.0 PL=0
MOVL C00603 V=800.0 PL=0
MOVL C00604 V=800.0 PL=0
MOVL C00605 V=800.0 PL=0
MOVL C00606 V=800.0 PL=0
MOVL C00607 V=800.0 PL=0
MOVL C00608 V=800.0 PL=0
MOVL C00609 V=800.0 PL=0
MOVL C00610 V=800.0 PL=0
MOVL C00611 V=800.0 PL=0
MOVL C00612 V=800.0 PL=0
MOVL C00613 V=800.0 PL=0
MOVL C00614 V=800.0 PL=0
MOVL C00615 V=800.0 PL=0
MOVL C00616 V=800.0 PL=0
MOVL C00617 V=800.0 PL=0
MOVL C00618 V=800.0 PL=0
MOVL C00619 V=800.0 PL=0
MOVL C00620 V=800.0 PL=0
MOVL C00621 V=800.0 PL=0
MOVL C00622 V=800.0 PL=0
MOVL C00623 V=800.0 PL=0
MOVL C00624 V=800.0 PL=0
MOVL C00625 V=800.0 PL=0
MOVL C00626 V=800.0 PL=0
MOVL C00627 V=800.0 PL=0
MOVL C00628 V=800.0 PL=0
MOVL C00629 V=800.0 PL=0
MOVL C00630 V=800.0 PL=0
MOVL C00631 V=800.0 PL=0
MOVL C00632 V=800.0 PL=0
MOVL C00633 V=800.0 PL=0
MOVL C00634 V=800.0 PL=0
MOVL C00635 V=800.0 PL=0
MOVL C00636 V=800.0 PL=0
MOVL C00637 V=800.0 PL=0
MOVL C00638 V=800.0 PL=0
MOVL C00639 V=800.0 PL=0
MOVL C00640 V=800.0 PL=0
MOVL C00641 V=800.0 PL=0
MOVL C00642 V=800.0 PL=0
MOVL C00643 V=800.0 PL=0
MOVL C00644 V=800.0 PL=0
MOVL C00645 V=800.0 PL=0
MOVL C00646 V=800.0 PL=0
MOVL C00647 V=800.0 PL=0
MOVL C00648 V=800.0 PL=0
MOVL C00649 V=800.0 PL=0
MOVL C00650 V=800.0 PL=0
MOVL C00651 V=800.0 PL=0
MOVL C00652 V=800.0 PL=0
MOVL C00653 V=800.0 PL=0
MOVL C00654 V=800.0 PL=0
MOVL C00655 V=800.0 PL=0
MOVL C00656 V=800.0 PL=0
MOVL C00657 V=800.0 PL=0
MOVL C00658 V=800.0 PL=0
MOVL C00659 V=800.0 PL=0
MOVL C00660 V=800.0 PL=0
MOVL C00661 V=800.0 PL=0
MOVL C00662 V=800.0 PL=0
MOVL C00663 V=800.0 PL=0
MOVL C00664 V=800.0 PL=0
MOVL C00665 V=800.0 PL=0
MOVL C00666 V=800.0 PL=0
MOVL C00667 V=800.0 PL=0
MOVL C00668 V=800.0 PL=0
MOVL C00669 V=800.0 PL=0
MOVL C00670 V=800.0 PL=0
MOVL C00671 V=800.0 PL=0
MOVL C00672 V=800.0 PL=0
MOVL C00673 V=800.0 PL=0
MOVL C00674 V=800.0 PL=0
MOVL C00675 V=800.0 PL=0
MOVL C00676 V=800.0 PL=0
MOVL C00677 V=800.0 PL=0
MOVL C00678 V=800.0 PL=0
MOVL C00679 V=800.0 PL=0
MOVL C00680 V=800.0 PL=0
MOVL C00681 V=800.0 PL=0
MOVL C00682 V=800.0 PL=0
MOVL C00683 V=800.0 PL=0
MOVL C00684 V=800.0 PL=0
MOVL C00685 V=800.0 PL=0
MOVL C00686 V=800.0 PL=0
MOVL C00687 V=800.0 PL=0
MOVL C00688 V=800.0 PL=0
MOVL C00689 V=800.0 PL=0
MOVL C00690 V=800.0 PL=0
MOVL C00691 V=800.0 PL=0
MOVL C00692 V=800.0 PL=0
MOVL C00693 V=800.0 PL=0
MOVL C00694 V=800.0 PL=0
MOVL C00695 V=800.0 PL=0
MOVL C00696 V=800.0 PL=0
MOVL C00697 V=800.0 PL=0
MOVL C00698 V=800.0 PL=0
MOVL C00699 V=800.0 PL=0
MOVL C00700 V=800.0 PL=0
MOVL C00701 V=800.0 PL=0
MOVL C00702 V=800.0 PL=0
MOVL C00703 V=800.0 PL=0
MOVL C00704 V=800.0 PL=0
MOVL C00705 V=800.0 PL=0
MOVL C00706 V=800.0 PL=0
MOVL C00707 V=800.0 PL=0
MOVL C00708 V=800.0 PL=0
MOVL C00709 V=800.0 PL=0
MOVL C00710 V=800.0 PL=0
MOVL C00711 V=800.0 PL=0
MOVL C00712 V=800.0 PL=0
MOVL C00713 V=800.0 PL=0
MOVL C00714 V=800.0 PL=0
MOVL C00715 V=800.0 PL=0
MOVL C00716 V=800.0 PL=0
MOVL C00717 V=800.0 PL=0
MOVL C00718 V=800.0 PL=0
MOVL C00719 V=800.0 PL=0
MOVL C00720 V=800.0 PL=0
MOVL C00721 V=800.0 PL=0
MOVL C00722 V=800.0 PL=0
MOVL C00723 V=800.0 PL=0
MOVL C00724 V=800.0 PL=0
MOVL C00725 V=800.0 PL=0
MOVL C00726 V=800.0 PL=0
MOVL C00727 V=800.0 PL=0
MOVL C00728 V=800.0 PL=0
MOVL C00729 V=800.0 PL=0
MOVL C00730 V=800.0 PL=0
MOVL C00731 V=800.0 PL=0
MOVL C00732 V=800.0 PL=0
MOVL C00733 V=800.0 PL=0
MOVL C00734 V=800.0 PL=0
MOVL C00735 V=800.0 PL=0
MOVL C00736 V=800.0 PL=0
MOVL C00737 V=800.0 PL=0
MOVL C00738 V=800.0 PL=0
MOVL C00739 V=800.0 PL=0
MOVL C00740 V=800.0 PL=0
MOVL C00741 V=800.0 PL=0
MOVL C00742 V=800.0 PL=0
MOVL C00743 V=800.0 PL=0
MOVL C00744 V=800.0 PL=0
MOVL C00745 V=800.0 PL=0
MOVL C00746 V=800.0 PL=0
MOVL C00747 V=800.0 PL=0
MOVL C00748 V=800.0 PL=0
MOVL C00749 V=800.0 PL=0
MOVL C00750 V=800.0 PL=0
MOVL C00751 V=800.0 PL=0
MOVL C00752 V=800.0 PL=0
MOVL C00753 V=800.0 PL=0
MOVL C00754 V=800.0 PL=0
MOVL C00755 V=800.0 PL=0
MOVL C00756 V=800.0 PL=0
MOVL C00757 V=800.0 PL=0
MOVL C00758 V=800.0 PL=0
MOVL C00759 V=800.0 PL=0
MOVL C00760 V=800.0 PL=0
MOVL C00761 V=800.0 PL=0
MOVL C00762 V=800.0 PL=0
MOVL C00763 V=800.0 PL=0
MOVL C00764 V=800.0 PL=0
MOVL C00765 V=800.0 PL=0
MOVL C00766 V=800.0 PL=0
MOVL C00767 V=800.0 PL=0
MOVL C00768 V=800.0 PL=0
MOVL C00769 V=800.0 PL=0
MOVL C00770 V=800.0 PL=0
MOVL C00771 V=800.0 PL=0
MOVL C00772 V=800.0 PL=0
MOVL C00773 V=800.0 PL=0
MOVL C00774 V=800.0 PL=0
MOVL C00775 V=800.0 PL=0
MOVL C00776 V=800.0 PL=0
MOVL C00777 V=800.0 PL=0
MOVL C00778 V=800.0 PL=0
MOVL C00779 V=800.0 PL=0
MOVL C00780 V=800.0 PL=0
MOVL C00781 V=800.0 PL=0
MOVL C00782 V=800.0 PL=0
MOVL C00783 V=800.0 PL=0
MOVL C00784 V=800.0 PL=0
MOVL C00785 V=800.0 PL=0
MOVL C00786 V=800.0 PL=0
MOVL C00787 V=800.0 PL=0
MOVL C00788 V=800.0 PL=0
MOVL C00789 V=800.0 PL=0
MOVL C00790 V=800.0 PL=0
MOVL C00791 V=800.0 PL=0
MOVL C00792 V=800.0 PL=0
MOVL C00793 V=800.0 PL=0
MOVL C00794 V=800.0 PL=0
MOVL C00795 V=800.0 PL=0
MOVL C00796 V=800.0 PL=0
MOVL C00797 V=800.0 PL=0
MOVL C00798 V=800.0 PL=0
MOVL C00799 V=800.0 PL=0
MOVL C00800 V=800.0 PL=0
MOVL C00801 V=800.0 PL=0
MOVL C00802 V=800.0 PL=0
MOVL C00803 V=800.0 PL=0
MOVL C00804 V=800.0 PL=0
MOVL C00805 V=800.0 PL=0
MOVL C00806 V=800.0 PL=0
MOVL C00807 V=800.0 PL=0
MOVL C00808 V=800.0 PL=0
MOVL C00809 V=800.0 PL=0
MOVL C00810 V=800.0 PL=0
MOVL C00811 V=800.0 PL=0
MOVL C00812 V=800.0 PL=0
MOVL C00813 V=800.0 PL=0
MOVL C00814 V=800.0 PL=0
MOVL C00815 V=800.0 PL=0
MOVL C00816 V=800.0 PL=0
MOVL C00817 V=800.0 PL=0
MOVL C00818 V=800.0 PL=0
MOVL C00819 V=800.0 PL=0
MOVL C00820 V=800.0 PL=0
MOVL C00821 V=800.0 PL=0
MOVL C00822 V=800.0 PL=0
MOVL C00823 V=800.0 PL=0
MOVL C00824 V=800.0 PL=0
MOVL C00825 V=800.0 PL=0
MOVL C00826 V=800.0 PL=0
MOVL C00827 V=800.0 PL=0
MOVL C00828 V=800.0 PL=0
MOVL C00829 V=800.0 PL=0
MOVL C00830 V=800.0 PL=0
MOVL C00831 V=800.0 PL=0
MOVL C00832 V=800.0 PL=0
MOVL C00833 V=800.0 PL=0
MOVL C00834 V=800.0 PL=0
MOVL C00835 V=800.0 PL=0
MOVL C00836 V=800.0 PL=0
MOVL C00837 V=800.0 PL=0
MOVL C00838 V=800.0 PL=0
MOVL C00839 V=800.0 PL=0
MOVL C00840 V=800.0 PL=0
MOVL C00841 V=800.0 PL=0
MOVL C00842 V=800.0 PL=0
MOVL C00843 V=800.0 PL=0
MOVL C00844 V=800.0 PL=0
MOVL C00845 V=800.0 PL=0
MOVL C00846 V=800.0 PL=0
MOVL C00847 V=800.0 PL=0
MOVL C00848 V=800.0 PL=0
MOVL C00849 V=800.0 PL=0
MOVL C00850 V=800.0 PL=0
MOVL C00851 V=800.0 PL=0
MOVL C00852 V=800.0 PL=0
MOVL C00853 V=800.0 PL=0
MOVL C00854 V=800.0 PL=0
MOVL C00855 V=800.0 PL=0
MOVL C00856 V=800.0 PL=0
MOVL C00857 V=800.0 PL=0
MOVL C00858 V=800.0 PL=0
MOVL C00859 V=800.0 PL=0
MOVL C00860 V=800.0 PL=0
MOVL C00861 V=800.0 PL=0
MOVL C00862 V=800.0 PL=0
MOVL C00863 V=800.0 PL=0
MOVL C00864 V=800.0 PL=0
MOVL C00865 V=800.0 PL=0
MOVL C00866 V=800.0 PL=0
MOVL C00867 V=800.0 PL=0
MOVL C00868 V=800.0 PL=0
MOVL C00869 V=800.0 PL=0
MOVL C00870 V=800.0 PL=0
MOVL C00871 V=800.0 PL=0
MOVL C00872 V=800.0 PL=0
MOVL C00873 V=800.0 PL=0
MOVL C00874 V=800.0 PL=0
MOVL C00875 V=800.0 PL=0
MOVL C00876 V=800.0 PL=0
MOVL C00877 V=800.0 PL=0
MOVL C00878 V=800.0 PL=0
MOVL C00879 V=800.0 PL=0
MOVL C00880 V=800.0 PL=0
MOVL C00881 V=800.0 PL=0
MOVL C00882 V=800.0 PL=0
MOVL C00883 V=800.0 PL=0
MOVL C00884 V=800.0 PL=0
MOVL C00885 V=800.0 PL=0
MOVL C00886 V=800.0 PL=0
MOVL C00887 V=800.0 PL=0
MOVL C00888 V=800.0 PL=0
MOVL C00889 V=800.0 PL=0
MOVL C00890 V=800.0 PL=0
MOVL C00891 V=800.0 PL=0
MOVL C00892 V=800.0 PL=0
MOVL C00893 V=800.0 PL=0
MOVL C00894 V=800.0 PL=0
MOVL C00895 V=800.0 PL=0
MOVL C00896 V=800.0 PL=0
MOVL C00897 V=800.0 PL=0
MOVL C00898 V=800.0 PL=0
MOVL C00899 V=800.0 PL=0
MOVL C00900 V=800.0 PL=0
MOVL C00901 V=800.0 PL=0
MOVL C00902 V=800.0 PL=0
MOVL C00903 V=800.0 PL=0
MOVL C00904 V=800.0 PL=0
MOVL C00905 V=800.0 PL=0
MOVL C00906 V=800.0 PL=0
MOVL C00907 V=800.0 PL=0
MOVL C00908 V=800.0 PL=0
MOVL C00909 V=800.0 PL=0
MOVL C00910 V=800.0 PL=0
MOVL C00911 V=800.0 PL=0
MOVL C00912 V=800.0 PL=0
MOVL C00913 V=800.0 PL=0
MOVL C00914 V=800.0 PL=0
MOVL C00915 V=800.0 PL=0
MOVL C00916 V=800.0 PL=0
MOVL C00917 V=800.0 PL=0
MOVL C00918 V=800.0 PL=0
MOVL C00919 V=800.0 PL=0
MOVL C00920 V=800.0 PL=0
MOVL C00921 V=800.0 PL=0
MOVL C00922 V=800.0 PL=0
MOVL C00923 V=800.0 PL=0
MOVL C00924 V=800.0 PL=0
MOVL C00925 V=800.0 PL=0
MOVL C00926 V=800.0 PL=0
MOVL C00927 V=800.0 PL=0
MOVL C00928 V=800.0 PL=0
MOVL C00929 V=800.0 PL=0
MOVL C00930 V=800.0 PL=0
MOVL C00931 V=800.0 PL=0
MOVL C00932 V=800.0 PL=0
MOVL C00933 V=800.0 PL=0
MOVL C00934 V=800.0 PL=0
MOVL C00935 V=800.0 PL=0
MOVL C00936 V=800.0 PL=0
MOVL C00937 V=800.0 PL=0
MOVL C00938 V=800.0 PL=0
MOVL C00939 V=800.0 PL=0
MOVL C00940 V=800.0 PL=0
MOVL C00941 V=800.0 PL=0
MOVL C00942 V=800.0 PL=0
MOVL C00943 V=800.0 PL=0
MOVL C00944 V=800.0 PL=0
MOVL C00945 V=800.0 PL=0
MOVL C00946 V=800.0 PL=0
MOVL C00947 V=800.0 PL=0
MOVL C00948 V=800.0 PL=0
MOVL C00949 V=800.0 PL=0
MOVL C00950 V=800.0 PL=0
MOVL C00951 V=800.0 PL=0
MOVL C00952 V=800.0 PL=0
MOVL C00953 V=800.0 PL=0
MOVL C00954 V=800.0 PL=0
MOVL C00955 V=800.0 PL=0
MOVL C00956 V=800.0 PL=0
MOVL C00957 V=800.0 PL=0
MOVL C00958 V=800.0 PL=0
MOVL C00959 V=800.0 PL=0
MOVL C00960 V=800.0 PL=0
MOVL C00961 V=800.0 PL=0
MOVL C00962 V=800.0 PL=0
MOVL C00963 V=800.0 PL=0
MOVL C00964 V=800.0 PL=0
MOVL C00965 V=800.0 PL=0
MOVL C00966 V=800.0 PL=0
MOVL C00967 V=800.0 PL=0
MOVL C00968 V=800.0 PL=0
MOVL C00969 V=800.0 PL=0
MOVL C00970 V=800.0 PL=0
MOVL C00971 V=800.0 PL=0
MOVL C00972 V=800.0 PL=0
MOVL C00973 V=800.0 PL=0
MOVL C00974 V=800.0 PL=0
MOVL C00975 V=800.0 PL=0
MOVL C00976 V=800.0 PL=0
MOVL C00977 V=800.0 PL=0
MOVL C00978 V=800.0 PL=0
MOVL C00979 V=800.0 PL=0
MOVL C00980 V=800.0 PL=0
MOVL C00981 V=800.0 PL=0
MOVL C00982 V=800.0 PL=0
MOVL C00983 V=800.0 PL=0
MOVL C00984 V=800.0 PL=0
MOVL C00985 V=800.0 PL=0
MOVL C00986 V=800.0 PL=0
MOVL C00987 V=800.0 PL=0
MOVL C00988 V=800.0 PL=0
MOVL C00989 V=800.0 PL=0
MOVL C00990 V=800.0 PL=0
MOVL C00991 V=800.0 PL=0
MOVL C00992 V=800.0 PL=0
MOVL C00993 V=800.0 PL=0
MOVL C00994 V=800.0 PL=0
MOVL C00995 V=800.0 PL=0
MOVL C00996 V=800.0 PL=0
MOVL C00997 V=800.0 PL=0
MOVL C00998 V=800.0 PL=0
MOVL C00999 V=800.0 PL=0
MOVL C01000 V=800.0 PL=0
MOVL C01001 V=800.0 PL=0
MOVL C01002 V=800.0 PL=0
MOVL C01003 V=800.0 PL=0
MOVL C01004 V=800.0 PL=0
MOVL C01005 V=800.0 PL=0
MOVL C01006 V=800.0 PL=0
MOVL C01007 V=800.0 PL=0
MOVL C01008 V=800.0 PL=0
MOVL C01009 V=800.0 PL=0
MOVL C01010 V=800.0 PL=0
MOVL C01011 V=800.0 PL=0
MOVL C01012 V=800.0 PL=0
MOVL C01013 V=800.0 PL=0
MOVL C01014 V=800.0 PL=0
MOVL C01015 V=800.0 PL=0
MOVL C01016 V=800.0 PL=0
MOVL C01017 V=800.0 PL=0
MOVL C01018 V=800.0 PL=0
MOVL C01019 V=800.0 PL=0
MOVL C01020 V=800.0 PL=0
MOVL C01021 V=800.0 PL=0
MOVL C01022 V=800.0 PL=0
MOVL C01023 V=800.0 PL=0
MOVL C01024 V=800.0 PL=0
MOVL C01025 V=800.0 PL=0
MOVL C01026 V=800.0 PL=0
MOVL C01027 V=800.0 PL=0
MOVL C01028 V=800.0 PL=0
MOVL C01029 V=800.0 PL=0
MOVL C01030 V=800.0 PL=0
MOVL C01031 V=800.0 PL=0
MOVL C01032 V=800.0 PL=0
MOVL C01033 V=800.0 PL=0
MOVL C01034 V=800.0 PL=0
MOVL C01035 V=800.0 PL=0
MOVL C01036 V=800.0 PL=0
MOVL C01037 V=800.0 PL=0
MOVL C01038 V=800.0 PL=0
MOVL C01039 V=800.0 PL=0
MOVL C01040 V=800.0 PL=0
MOVL C01041 V=800.0 PL=0
MOVL C01042 V=800.0 PL=0
MOVL C01043 V=800.0 PL=0
MOVL C01044 V=800.0 PL=0
MOVL C01045 V=800.0 PL=0
MOVL C01046 V=800.0 PL=0
MOVL C01047 V=800.0 PL=0
MOVL C01048 V=800.0 PL=0
MOVL C01049 V=800.0 PL=0
MOVL C01050 V=800.0 PL=0
MOVL C01051 V=800.0 PL=0
MOVL C01052 V=800.0 PL=0
MOVL C01053 V=800.0 PL=0
MOVL C01054 V=800.0 PL=0
MOVL C01055 V=800.0 PL=0
MOVL C01056 V=800.0 PL=0
MOVL C01057 V=800.0 PL=0
MOVL C01058 V=800.0 PL=0
MOVL C01059 V=800.0 PL=0
MOVL C01060 V=800.0 PL=0
MOVL C01061 V=800.0 PL=0
MOVL C01062 V=800.0 PL=0
MOVL C01063 V=800.0 PL=0
MOVL C01064 V=800.0 PL=0
MOVL C01065 V=800.0 PL=0
MOVL C01066 V=800.0 PL=0
MOVL C01067 V=800.0 PL=0
MOVL C01068 V=800.0 PL=0
MOVL C01069 V=800.0 PL=0
MOVL C01070 V=800.0 PL=0
MOVL C01071 V=800.0 PL=0
MOVL C01072 V=800.0 PL=0
MOVL C01073 V=800.0 PL=0
MOVL C01074 V=800.0 PL=0
MOVL C01075 V=800.0 PL=0
MOVL C01076 V=800.0 PL=0
MOVL C01077 V=800.0 PL=0
MOVL C01078 V=800.0 PL=0
MOVL C01079 V=800.0 PL=0
MOVL C01080 V=800.0 PL=0
MOVL C01081 V=800.0 PL=0
MOVL C01082 V=800.0 PL=0
MOVL C01083 V=800.0 PL=0
MOVL C01084 V=800.0 PL=0
MOVL C01085 V=800.0 PL=0
MOVL C01086 V=800.0 PL=0
MOVL C01087 V=800.0 PL=0
MOVL C01088 V=800.0 PL=0
MOVL C01089 V=800.0 PL=0
MOVL C01090 V=800.0 PL=0
MOVL C01091 V=800.0 PL=0
MOVL C01092 V=800.0 PL=0
MOVL C01093 V=800.0 PL=0
MOVL C01094 V=800.0 PL=0
MOVL C01095 V=800.0 PL=0
MOVL C01096 V=800.0 PL=0
MOVL C01097 V=800.0 PL=0
MOVL C01098 V=800.0 PL=0
MOVL C01099 V=800.0 PL=0
MOVL C01100 V=800.0 PL=0
MOVL C01101 V=800.0 PL=0
MOVL C01102 V=800.0 PL=0
MOVL C01103 V=800.0 PL=0
MOVL C01104 V=800.0 PL=0
MOVL C01105 V=800.0 PL=0
MOVL C01106 V=800.0 PL=0
MOVL C01107 V=800.0 PL=0
MOVL C01108 V=800.0 PL=0
MOVL C01109 V=800.0 PL=0
MOVL C01110 V=800.0 PL=0
MOVL C01111 V=800.0 PL=0
MOVL C01112 V=800.0 PL=0
MOVL C01113 V=800.0 PL=0
MOVL C01114 V=800.0 PL=0
MOVL C01115 V=800.0 PL=0
MOVL C01116 V=800.0 PL=0
MOVL C01117 V=800.0 PL=0
MOVL C01118 V=800.0 PL=0
MOVL C01119 V=800.0 PL=0
MOVL C01120 V=800.0 PL=0
MOVL C01121 V=800.0 PL=0
MOVL C01122 V=800.0 PL=0
MOVL C01123 V=800.0 PL=0
MOVL C01124 V=800.0 PL=0
MOVL C01125 V=800.0 PL=0
MOVL C01126 V=800.0 PL=0
MOVL C01127 V=800.0 PL=0
MOVL C01128 V=800.0 PL=0
MOVL C01129 V=800.0 PL=0
MOVL C01130 V=800.0 PL=0
MOVL C01131 V=800.0 PL=0
MOVL C01132 V=800.0 PL=0
MOVL C01133 V=800.0 PL=0
MOVL C01134 V=800.0 PL=0
MOVL C01135 V=800.0 PL=0
MOVL C01136 V=800.0 PL=0
MOVL C01137 V=800.0 PL=0
MOVL C01138 V=800.0 PL=0
MOVL C01139 V=800.0 PL=0
MOVL C01140 V=800.0 PL=0
MOVL C01141 V=800.0 PL=0
MOVL C01142 V=800.0 PL=0
MOVL C01143 V=800.0 PL=0
MOVL C01144 V=800.0 PL=0
MOVL C01145 V=800.0 PL=0
MOVL C01146 V=800.0 PL=0
MOVL C01147 V=800.0 PL=0
MOVL C01148 V=800.0 PL=0
MOVL C01149 V=800.0 PL=0
MOVL C01150 V=800.0 PL=0
MOVL C01151 V=800.0 PL=0
MOVL C01152 V=800.0 PL=0
MOVL C01153 V=800.0 PL=0
MOVL C01154 V=800.0 PL=0
MOVL C01155 V=800.0 PL=0
MOVL C01156 V=800.0 PL=0
MOVL C01157 V=800.0 PL=0
MOVL C01158 V=800.0 PL=0
MOVL C01159 V=800.0 PL=0
MOVL C01160 V=800.0 PL=0
MOVL C01161 V=800.0 PL=0
MOVL C01162 V=800.0 PL=0
MOVL C01163 V=800.0 PL=0
MOVL C01164 V=800.0 PL=0
MOVL C01165 V=800.0 PL=0
MOVL C01166 V=800.0 PL=0
MOVL C01167 V=800.0 PL=0
MOVL C01168 V=800.0 PL=0
MOVL C01169 V=800.0 PL=0
MOVL C01170 V=800.0 PL=0
MOVL C01171 V=800.0 PL=0
MOVL C01172 V=800.0 PL=0
MOVL C01173 V=800.0 PL=0
MOVL C01174 V=800.0 PL=0
MOVL C01175 V=800.0 PL=0
MOVL C01176 V=800.0 PL=0
MOVL C01177 V=800.0 PL=0
MOVL C01178 V=800.0 PL=0
MOVL C01179 V=800.0 PL=0
MOVL C01180 V=800.0 PL=0
MOVL C01181 V=800.0 PL=0
MOVL C01182 V=800.0 PL=0
MOVL C01183 V=800.0 PL=0
MOVL C01184 V=800.0 PL=0
MOVL C01185 V=800.0 PL=0
MOVL C01186 V=800.0 PL=0
MOVL C01187 V=800.0 PL=0
MOVL C01188 V=800.0 PL=0
MOVL C01189 V=800.0 PL=0
MOVL C01190 V=800.0 PL=0
MOVL C01191 V=800.0 PL=0
MOVL C01192 V=800.0 PL=0
MOVL C01193 V=800.0 PL=0
MOVL C01194 V=800.0 PL=0
MOVL C01195 V=800.0 PL=0
MOVL C01196 V=800.0 PL=0
MOVL C01197 V=800.0 PL=0
MOVL C01198 V=800.0 PL=0
MOVL C01199 V=800.0 PL=0
MOVL C01200 V=800.0 PL=0
MOVL C01201 V=800.0 PL=0
MOVL C01202 V=800.0 PL=0
MOVL C01203 V=800.0 PL=0
MOVL C01204 V=800.0 PL=0
MOVL C01205 V=800.0 PL=0
MOVL C01206 V=800.0 PL=0
MOVL C01207 V=800.0 PL=0
MOVL C01208 V=800.0 PL=0
MOVL C01209 V=800.0 PL=0
MOVL C01210 V=800.0 PL=0
MOVL C01211 V=800.0 PL=0
MOVL C01212 V=800.0 PL=0
MOVL C01213 V=800.0 PL=0
MOVL C01214 V=800.0 PL=0
MOVL C01215 V=800.0 PL=0
MOVL C01216 V=800.0 PL=0
MOVL C01217 V=800.0 PL=0
MOVL C01218 V=800.0 PL=0
MOVL C01219 V=800.0 PL=0
MOVL C01220 V=800.0 PL=0
MOVL C01221 V=800.0 PL=0
MOVL C01222 V=800.0 PL=0
MOVL C01223 V=800.0 PL=0
MOVL C01224 V=800.0 PL=0
MOVL C01225 V=800.0 PL=0
MOVL C01226 V=800.0 PL=0
MOVL C01227 V=800.0 PL=0
MOVL C01228 V=800.0 PL=0
MOVL C01229 V=800.0 PL=0
MOVL C01230 V=800.0 PL=0
MOVL C01231 V=800.0 PL=0
MOVL C01232 V=800.0 PL=0
MOVL C01233 V=800.0 PL=0
MOVL C01234 V=800.0 PL=0
MOVL C01235 V=800.0 PL=0
MOVL C01236 V=800.0 PL=0
MOVL C01237 V=800.0 PL=0
MOVL C01238 V=800.0 PL=0
MOVL C01239 V=800.0 PL=0
MOVL C01240 V=800.0 PL=0
MOVL C01241 V=800.0 PL=0
MOVL C01242 V=800.0 PL=0
MOVL C01243 V=800.0 PL=0
MOVL C01244 V=800.0 PL=0
MOVL C01245 V=800.0 PL=0
MOVL C01246 V=800.0 PL=0
MOVL C01247 V=800.0 PL=0
MOVL C01248 V=800.0 PL=0
MOVL C01249 V=800.0 PL=0
MOVL C01250 V=800.0 PL=0
MOVL C01251 V=800.0 PL=0
MOVL C01252 V=800.0 PL=0
MOVL C01253 V=800.0 PL=0
MOVL C01254 V=800.0 PL=0
MOVL C01255 V=800.0 PL=0
MOVL C01256 V=800.0 PL=0
MOVL C01257 V=800.0 PL=0
MOVL C01258 V=800.0 PL=0
MOVL C01259 V=800.0 PL=0
MOVL C01260 V=800.0 PL=0
MOVL C01261 V=800.0 PL=0
MOVL C01262 V=800.0 PL=0
MOVL C01263 V=800.0 PL=0
MOVL C01264 V=800.0 PL=0
MOVL C01265 V=800.0 PL=0
MOVL C01266 V=800.0 PL=0
MOVL C01267 V=800.0 PL=0
MOVL C01268 V=800.0 PL=0
MOVL C01269 V=800.0 PL=0
MOVL C01270 V=800.0 PL=0
MOVL C01271 V=800.0 PL=0
MOVL C01272 V=800.0 PL=0
MOVL C01273 V=800.0 PL=0
MOVL C01274 V=800.0 PL=0
MOVL C01275 V=800.0 PL=0
MOVL C01276 V=800.0 PL=0
MOVL C01277 V=800.0 PL=0
MOVL C01278 V=800.0 PL=0
MOVL C01279 V=800.0 PL=0
MOVL C01280 V=800.0 PL=0
MOVL C01281 V=800.0 PL=0
MOVL C01282 V=800.0 PL=0
MOVL C01283 V=800.0 PL=0
MOVL C01284 V=800.0 PL=0
MOVL C01285 V=800.0 PL=0
MOVL C01286 V=800.0 PL=0
MOVL C01287 V=800.0 PL=0
MOVL C01288 V=800.0 PL=0
MOVL C01289 V=800.0 PL=0
MOVL C01290 V=800.0 PL=0
MOVL C01291 V=800.0 PL=0
MOVL C01292 V=800.0 PL=0
MOVL C01293 V=800.0 PL=0
MOVL C01294 V=800.0 PL=0
MOVL C01295 V=800.0 PL=0
MOVL C01296 V=800.0 PL=0
MOVL C01297 V=800.0 PL=0
MOVL C01298 V=800.0 PL=0
MOVL C01299 V=800.0 PL=0
MOVL C01300 V=800.0 PL=0
MOVL C01301 V=800.0 PL=0
MOVL C01302 V=800.0 PL=0
MOVL C01303 V=800.0 PL=0
MOVL C01304 V=800.0 PL=0
MOVL C01305 V=800.0 PL=0
MOVL C01306 V=800.0 PL=0
MOVL C01307 V=800.0 PL=0
MOVL C01308 V=800.0 PL=0
MOVL C01309 V=800.0 PL=0
MOVL C01310 V=800.0 PL=0
MOVL C01311 V=800.0 PL=0
MOVL C01312 V=800.0 PL=0
MOVL C01313 V=800.0 PL=0
MOVL C01314 V=800.0 PL=0
MOVL C01315 V=800.0 PL=0
MOVL C01316 V=800.0 PL=0
MOVL C01317 V=800.0 PL=0
MOVL C01318 V=800.0 PL=0
MOVL C01319 V=800.0 PL=0
MOVL C01320 V=800.0 PL=0
MOVL C01321 V=800.0 PL=0
MOVL C01322 V=800.0 PL=0
MOVL C01323 V=800.0 PL=0
MOVL C01324 V=800.0 PL=0
MOVL C01325 V=800.0 PL=0
MOVL C01326 V=800.0 PL=0
MOVL C01327 V=800.0 PL=0
MOVL C01328 V=800.0 PL=0
MOVL C01329 V=800.0 PL=0
MOVL C01330 V=800.0 PL=0
MOVL C01331 V=800.0 PL=0
MOVL C01332 V=800.0 PL=0
MOVL C01333 V=800.0 PL=0
MOVL C01334 V=800.0 PL=0
MOVL C01335 V=800.0 PL=0
MOVL C01336 V=800.0 PL=0
MOVL C01337 V=800.0 PL=0
MOVL C01338 V=800.0 PL=0
MOVL C01339 V=800.0 PL=0
MOVL C01340 V=800.0 PL=0
MOVL C01341 V=800.0 PL=0
MOVL C01342 V=800.0 PL=0
MOVL C01343 V=800.0 PL=0
MOVL C01344 V=800.0 PL=0
MOVL C01345 V=800.0 PL=0
MOVL C01346 V=800.0 PL=0
MOVL C01347 V=800.0 PL=0
MOVL C01348 V=800.0 PL=0
MOVL C01349 V=800.0 PL=0
MOVL C01350 V=800.0 PL=0
MOVL C01351 V=800.0 PL=0
MOVL C01352 V=800.0 PL=0
MOVL C01353 V=800.0 PL=0
MOVL C01354 V=800.0 PL=0
MOVL C01355 V=800.0 PL=0
MOVL C01356 V=800.0 PL=0
MOVL C01357 V=800.0 PL=0
MOVL C01358 V=800.0 PL=0
MOVL C01359 V=800.0 PL=0
MOVL C01360 V=800.0 PL=0
MOVL C01361 V=800.0 PL=0
MOVL C01362 V=800.0 PL=0
MOVL C01363 V=800.0 PL=0
MOVL C01364 V=800.0 PL=0
MOVL C01365 V=800.0 PL=0
MOVL C01366 V=800.0 PL=0
MOVL C01367 V=800.0 PL=0
MOVL C01368 V=800.0 PL=0
MOVL C01369 V=800.0 PL=0
MOVL C01370 V=800.0 PL=0
MOVL C01371 V=800.0 PL=0
MOVL C01372 V=800.0 PL=0
MOVL C01373 V=800.0 PL=0
MOVL C01374 V=800.0 PL=0
MOVL C01375 V=800.0 PL=0
MOVL C01376 V=800.0 PL=0
MOVL C01377 V=800.0 PL=0
MOVL C01378 V=800.0 PL=0
MOVL C01379 V=800.0 PL=0
MOVL C01380 V=800.0 PL=0
MOVL C01381 V=800.0 PL=0
MOVL C01382 V=800.0 PL=0
MOVL C01383 V=800.0 PL=0
MOVL C01384 V=800.0 PL=0
MOVL C01385 V=800.0 PL=0
MOVL C01386 V=800.0 PL=0
MOVL C01387 V=800.0 PL=0
MOVL C01388 V=800.0 PL=0
MOVL C01389 V=800.0 PL=0
MOVL C01390 V=800.0 PL=0
MOVL C01391 V=800.0 PL=0
MOVL C01392 V=800.0 PL=0
MOVL C01393 V=800.0 PL=0
MOVL C01394 V=800.0 PL=0
MOVL C01395 V=800.0 PL=0
MOVL C01396 V=800.0 PL=0
MOVL C01397 V=800.0 PL=0
MOVL C01398 V=800.0 PL=0
MOVL C01399 V=800.0 PL=0
MOVL C01400 V=800.0 PL=0
MOVL C01401 V=800.0 PL=0
MOVL C01402 V=800.0 PL=0
MOVL C01403 V=800.0 PL=0
MOVL C01404 V=800.0 PL=0
MOVL C01405 V=800.0 PL=0
MOVL C01406 V=800.0 PL=0
MOVL C01407 V=800.0 PL=0
MOVL C01408 V=800.0 PL=0
MOVL C01409 V=800.0 PL=0
MOVL C01410 V=800.0 PL=0
MOVL C01411 V=800.0 PL=0
MOVL C01412 V=800.0 PL=0
MOVL C01413 V=800.0 PL=0
MOVL C01414 V=800.0 PL=0
MOVL C01415 V=800.0 PL=0
MOVL C01416 V=800.0 PL=0
MOVL C01417 V=800.0 PL=0
MOVL C01418 V=800.0 PL=0
MOVL C01419 V=800.0 PL=0
MOVL C01420 V=800.0 PL=0
MOVL C01421 V=800.0 PL=0
MOVL C01422 V=800.0 PL=0
MOVL C01423 V=800.0 PL=0
MOVL C01424 V=800.0 PL=0
MOVL C01425 V=800.0 PL=0
MOVL C01426 V=800.0 PL=0
MOVL C01427 V=800.0 PL=0
MOVL C01428 V=800.0 PL=0
MOVL C01429 V=800.0 PL=0
MOVL C01430 V=800.0 PL=0
MOVL C01431 V=800.0 PL=0
MOVL C01432 V=800.0 PL=0
MOVL C01433 V=800.0 PL=0
MOVL C01434 V=800.0 PL=0
MOVL C01435 V=800.0 PL=0
MOVL C01436 V=800.0 PL=0
MOVL C01437 V=800.0 PL=0
MOVL C01438 V=800.0 PL=0
MOVL C01439 V=800.0 PL=0
MOVL C01440 V=800.0 PL=0
MOVL C01441 V=800.0 PL=0
MOVL C01442 V=800.0 PL=0
MOVL C01443 V=800.0 PL=0
MOVL C01444 V=800.0 PL=0
MOVL C01445 V=800.0 PL=0
MOVL C01446 V=800.0 PL=0
MOVL C01447 V=800.0 PL=0
MOVL C01448 V=800.0 PL=0
MOVL C01449 V=800.0 PL=0
MOVL C01450 V=800.0 PL=0
MOVL C01451 V=800.0 PL=0
MOVL C01452 V=800.0 PL=0
MOVL C01453 V=800.0 PL=0
MOVL C01454 V=800.0 PL=0
MOVL C01455 V=800.0 PL=0
MOVL C01456 V=800.0 PL=0
MOVL C01457 V=800.0 PL=0
MOVL C01458 V=800.0 PL=0
MOVL C01459 V=800.0 PL=0
MOVL C01460 V=800.0 PL=0
MOVL C01461 V=800.0 PL=0
MOVL C01462 V=800.0 PL=0
MOVL C01463 V=800.0 PL=0
MOVL C01464 V=800.0 PL=0
MOVL C01465 V=800.0 PL=0
MOVL C01466 V=800.0 PL=0
MOVL C01467 V=800.0 PL=0
MOVL C01468 V=800.0 PL=0
MOVL C01469 V=800.0 PL=0
MOVL C01470 V=800.0 PL=0
MOVL C01471 V=800.0 PL=0
MOVL C01472 V=800.0 PL=0
MOVL C01473 V=800.0 PL=0
MOVL C01474 V=800.0 PL=0
MOVL C01475 V=800.0 PL=0
MOVL C01476 V=800.0 PL=0
MOVL C01477 V=800.0 PL=0
MOVL C01478 V=800.0 PL=0
MOVL C01479 V=800.0 PL=0
MOVL C01480 V=800.0 PL=0
MOVL C01481 V=800.0 PL=0
MOVL C01482 V=800.0 PL=0
MOVL C01483 V=800.0 PL=0
MOVL C01484 V=800.0 PL=0
MOVL C01485 V=800.0 PL=0
MOVL C01486 V=800.0 PL=0
MOVL C01487 V=800.0 PL=0
MOVL C01488 V=800.0 PL=0
MOVL C01489 V=800.0 PL=0
MOVL C01490 V=800.0 PL=0
MOVL C01491 V=800.0 PL=0
MOVL C01492 V=800.0 PL=0
MOVL C01493 V=800.0 PL=0
MOVL C01494 V=800.0 PL=0
MOVL C01495 V=800.0 PL=0
MOVL C01496 V=800.0 PL=0
MOVL C01497 V=800.0 PL=0
MOVL C01498 V=800.0 PL=0
MOVL C01499 V=800.0 PL=0
MOVL C01500 V=800.0 PL=0
MOVL C01501 V=800.0 PL=0
MOVL C01502 V=800.0 PL=0
MOVL C01503 V=800.0 PL=0
MOVL C01504 V=800.0 PL=0
MOVL C01505 V=800.0 PL=0
MOVL C01506 V=800.0 PL=0
MOVL C01507 V=800.0 PL=0
MOVL C01508 V=800.0 PL=0
MOVL C01509 V=800.0 PL=0
MOVL C01510 V=800.0 PL=0
MOVL C01511 V=800.0 PL=0
MOVL C01512 V=800.0 PL=0
MOVL C01513 V=800.0 PL=0
MOVL C01514 V=800.0 PL=0
MOVL C01515 V=800.0 PL=0
MOVL C01516 V=800.0 PL=0
MOVL C01517 V=800.0 PL=0
MOVL C01518 V=800.0 PL=0
MOVL C01519 V=800.0 PL=0
MOVL C01520 V=800.0 PL=0
MOVL C01521 V=800.0 PL=0
MOVL C01522 V=800.0 PL=0
MOVL C01523 V=800.0 PL=0
MOVL C01524 V=800.0 PL=0
MOVL C01525 V=800.0 PL=0
MOVL C01526 V=800.0 PL=0
MOVL C01527 V=800.0 PL=0
MOVL C01528 V=800.0 PL=0
MOVL C01529 V=800.0 PL=0
MOVL C01530 V=800.0 PL=0
MOVL C01531 V=800.0 PL=0
MOVL C01532 V=800.0 PL=0
MOVL C01533 V=800.0 PL=0
MOVL C01534 V=800.0 PL=0
MOVL C01535 V=800.0 PL=0
MOVL C01536 V=800.0 PL=0
MOVL C01537 V=800.0 PL=0
MOVL C01538 V=800.0 PL=0
MOVL C01539 V=800.0 PL=0
MOVL C01540 V=800.0 PL=0
MOVL C01541 V=800.0 PL=0
MOVL C01542 V=800.0 PL=0
MOVL C01543 V=800.0 PL=0
MOVL C01544 V=800.0 PL=0
MOVL C01545 V=800.0 PL=0
MOVL C01546 V=800.0 PL=0
MOVL C01547 V=800.0 PL=0
MOVL C01548 V=800.0 PL=0
MOVL C01549 V=800.0 PL=0
MOVL C01550 V=800.0 PL=0
MOVL C01551 V=800.0 PL=0
MOVL C01552 V=800.0 PL=0
MOVL C01553 V=800.0 PL=0
MOVL C01554 V=800.0 PL=0
MOVL C01555 V=800.0 PL=0
MOVL C01556 V=800.0 PL=0
MOVL C01557 V=800.0 PL=0
MOVL C01558 V=800.0 PL=0
MOVL C01559 V=800.0 PL=0
MOVL C01560 V=800.0 PL=0
MOVL C01561 V=800.0 PL=0
MOVL C01562 V=800.0 PL=0
MOVL C01563 V=800.0 PL=0
MOVL C01564 V=800.0 PL=0
MOVL C01565 V=800.0 PL=0
MOVL C01566 V=800.0 PL=0
MOVL C01567 V=800.0 PL=0
MOVL C01568 V=800.0 PL=0
MOVL C01569 V=800.0 PL=0
MOVL C01570 V=800.0 PL=0
MOVL C01571 V=800.0 PL=0
MOVL C01572 V=800.0 PL=0
MOVL C01573 V=800.0 PL=0
MOVL C01574 V=800.0 PL=0
MOVL C01575 V=800.0 PL=0
MOVL C01576 V=800.0 PL=0
MOVL C01577 V=800.0 PL=0
MOVL C01578 V=800.0 PL=0
MOVL C01579 V=800.0 PL=0
MOVL C01580 V=800.0 PL=0
MOVL C01581 V=800.0 PL=0
MOVL C01582 V=800.0 PL=0
MOVL C01583 V=800.0 PL=0
MOVL C01584 V=800.0 PL=0
MOVL C01585 V=800.0 PL=0
MOVL C01586 V=800.0 PL=0
MOVL C01587 V=800.0 PL=0
MOVL C01588 V=800.0 PL=0
MOVL C01589 V=800.0 PL=0
MOVL C01590 V=800.0 PL=0
MOVL C01591 V=800.0 PL=0
MOVL C01592 V=800.0 PL=0
MOVL C01593 V=800.0 PL=0
MOVL C01594 V=800.0 PL=0
MOVL C01595 V=800.0 PL=0
MOVL C01596 V=800.0 PL=0
MOVL C01597 V=800.0 PL=0
MOVL C01598 V=800.0 PL=0
MOVL C01599 V=800.0 PL=0
MOVL C01600 V=800.0 PL=0
MOVL C01601 V=800.0 PL=0
MOVL C01602 V=800.0 PL=0
MOVL C01603 V=800.0 PL=0
MOVL C01604 V=800.0 PL=0
MOVL C01605 V=800.0 PL=0
MOVL C01606 V=800.0 PL=0
MOVL C01607 V=800.0 PL=0
MOVL C01608 V=800.0 PL=0
MOVL C01609 V=800.0 PL=0
MOVL C01610 V=800.0 PL=0
MOVL C01611 V=800.0 PL=0
MOVL C01612 V=800.0 PL=0
MOVL C01613 V=800.0 PL=0
MOVL C01614 V=800.0 PL=0
MOVL C01615 V=800.0 PL=0
MOVL C01616 V=800.0 PL=0
MOVL C01617 V=800.0 PL=0
MOVL C01618 V=800.0 PL=0
MOVL C01619 V=800.0 PL=0
MOVL C01620 V=800.0 PL=0
MOVL C01621 V=800.0 PL=0
MOVL C01622 V=800.0 PL=0
MOVL C01623 V=800.0 PL=0
MOVL C01624 V=800.0 PL=0
MOVL C01625 V=800.0 PL=0
MOVL C01626 V=800.0 PL=0
MOVL C01627 V=800.0 PL=0
MOVL C01628 V=800.0 PL=0
MOVL C01629 V=800.0 PL=0
MOVL C01630 V=800.0 PL=0
MOVL C01631 V=800.0 PL=0
MOVL C01632 V=800.0 PL=0
MOVL C01633 V=800.0 PL=0
MOVL C01634 V=800.0 PL=0
MOVL C01635 V=800.0 PL=0
MOVL C01636 V=800.0 PL=0
MOVL C01637 V=800.0 PL=0
MOVL C01638 V=800.0 PL=0
MOVL C01639 V=800.0 PL=0
MOVL C01640 V=800.0 PL=0
MOVL C01641 V=800.0 PL=0
MOVL C01642 V=800.0 PL=0
MOVL C01643 V=800.0 PL=0
MOVL C01644 V=800.0 PL=0
MOVL C01645 V=800.0 PL=0
MOVL C01646 V=800.0 PL=0
MOVL C01647 V=800.0 PL=0
MOVL C01648 V=800.0 PL=0
MOVL C01649 V=800.0 PL=0
MOVL C01650 V=800.0 PL=0
MOVL C01651 V=800.0 PL=0
MOVL C01652 V=800.0 PL=0
MOVL C01653 V=800.0 PL=0
MOVL C01654 V=800.0 PL=0
MOVL C01655 V=800.0 PL=0
MOVL C01656 V=800.0 PL=0
MOVL C01657 V=800.0 PL=0
MOVL C01658 V=800.0 PL=0
MOVL C01659 V=800.0 PL=0
MOVL C01660 V=800.0 PL=0
MOVL C01661 V=800.0 PL=0
MOVL C01662 V=800.0 PL=0
MOVL C01663 V=800.0 PL=0
MOVL C01664 V=800.0 PL=0
MOVL C01665 V=800.0 PL=0
MOVL C01666 V=800.0 PL=0
MOVL C01667 V=800.0 PL=0
MOVL C01668 V=800.0 PL=0
MOVL C01669 V=800.0 PL=0
MOVL C01670 V=800.0 PL=0
MOVL C01671 V=800.0 PL=0
MOVL C01672 V=800.0 PL=0
MOVL C01673 V=800.0 PL=0
MOVL C01674 V=800.0 PL=0
MOVL C01675 V=800.0 PL=0
MOVL C01676 V=800.0 PL=0
MOVL C01677 V=800.0 PL=0
MOVL C01678 V=800.0 PL=0
MOVL C01679 V=800.0 PL=0
MOVL C01680 V=800.0 PL=0
MOVL C01681 V=800.0 PL=0
MOVL C01682 V=800.0 PL=0
MOVL C01683 V=800.0 PL=0
MOVL C01684 V=800.0 PL=0
MOVL C01685 V=800.0 PL=0
MOVL C01686 V=800.0 PL=0
MOVL C01687 V=800.0 PL=0
MOVL C01688 V=800.0 PL=0
MOVL C01689 V=800.0 PL=0
MOVL C01690 V=800.0 PL=0
MOVL C01691 V=800.0 PL=0
MOVL C01692 V=800.0 PL=0
MOVL C01693 V=800.0 PL=0
MOVL C01694 V=800.0 PL=0
MOVL C01695 V=800.0 PL=0
MOVL C01696 V=800.0 PL=0
MOVL C01697 V=800.0 PL=0
MOVL C01698 V=800.0 PL=0
MOVL C01699 V=800.0 PL=0
MOVL C01700 V=800.0 PL=0
MOVL C01701 V=800.0 PL=0
MOVL C01702 V=800.0 PL=0
MOVL C01703 V=800.0 PL=0
MOVL C01704 V=800.0 PL=0
MOVL C01705 V=800.0 PL=0
MOVL C01706 V=800.0 PL=0
MOVL C01707 V=800.0 PL=0
MOVL C01708 V=800.0 PL=0
MOVL C01709 V=800.0 PL=0
MOVL C01710 V=800.0 PL=0
MOVL C01711 V=800.0 PL=0
MOVL C01712 V=800.0 PL=0
MOVL C01713 V=800.0 PL=0
MOVL C01714 V=800.0 PL=0
MOVL C01715 V=800.0 PL=0
MOVL C01716 V=800.0 PL=0
MOVL C01717 V=800.0 PL=0
MOVL C01718 V=800.0 PL=0
MOVL C01719 V=800.0 PL=0
MOVL C01720 V=800.0 PL=0
MOVL C01721 V=800.0 PL=0
MOVL C01722 V=800.0 PL=0
MOVL C01723 V=800.0 PL=0
MOVL C01724 V=800.0 PL=0
MOVL C01725 V=800.0 PL=0
MOVL C01726 V=800.0 PL=0
MOVL C01727 V=800.0 PL=0
MOVL C01728 V=800.0 PL=0
MOVL C01729 V=800.0 PL=0
MOVL C01730 V=800.0 PL=0
MOVL C01731 V=800.0 PL=0
MOVL C01732 V=800.0 PL=0
MOVL C01733 V=800.0 PL=0
MOVL C01734 V=800.0 PL=0
MOVL C01735 V=800.0 PL=0
MOVL C01736 V=800.0 PL=0
MOVL C01737 V=800.0 PL=0
MOVL C01738 V=800.0 PL=0
MOVL C01739 V=800.0 PL=0
MOVL C01740 V=800.0 PL=0
MOVL C01741 V=800.0 PL=0
MOVL C01742 V=800.0 PL=0
MOVL C01743 V=800.0 PL=0
MOVL C01744 V=800.0 PL=0
MOVL C01745 V=800.0 PL=0
MOVL C01746 V=800.0 PL=0
MOVL C01747 V=800.0 PL=0
MOVL C01748 V=800.0 PL=0
MOVL C01749 V=800.0 PL=0
MOVL C01750 V=800.0 PL=0
MOVL C01751 V=800.0 PL=0
MOVL C01752 V=800.0 PL=0
MOVL C01753 V=800.0 PL=0
MOVL C01754 V=800.0 PL=0
MOVL C01755 V=800.0 PL=0
MOVL C01756 V=800.0 PL=0
MOVL C01757 V=800.0 PL=0
MOVL C01758 V=800.0 PL=0
MOVL C01759 V=800.0 PL=0
MOVL C01760 V=800.0 PL=0
MOVL C01761 V=800.0 PL=0
MOVL C01762 V=800.0 PL=0
MOVL C01763 V=800.0 PL=0
MOVL C01764 V=800.0 PL=0
MOVL C01765 V=800.0 PL=0
MOVL C01766 V=800.0 PL=0
MOVL C01767 V=800.0 PL=0
MOVL C01768 V=800.0 PL=0
MOVL C01769 V=800.0 PL=0
MOVL C01770 V=800.0 PL=0
MOVL C01771 V=800.0 PL=0
MOVL C01772 V=800.0 PL=0
MOVL C01773 V=800.0 PL=0
MOVL C01774 V=800.0 PL=0
MOVL C01775 V=800.0 PL=0
MOVL C01776 V=800.0 PL=0
MOVL C01777 V=800.0 PL=0
MOVL C01778 V=800.0 PL=0
MOVL C01779 V=800.0 PL=0
MOVL C01780 V=800.0 PL=0
MOVL C01781 V=800.0 PL=0
MOVL C01782 V=800.0 PL=0
MOVL C01783 V=800.0 PL=0
MOVL C01784 V=800.0 PL=0
MOVL C01785 V=800.0 PL=0
MOVL C01786 V=800.0 PL=0
MOVL C01787 V=800.0 PL=0
MOVL C01788 V=800.0 PL=0
MOVL C01789 V=800.0 PL=0
MOVL C01790 V=800.0 PL=0
MOVL C01791 V=800.0 PL=0
MOVL C01792 V=800.0 PL=0
MOVL C01793 V=800.0 PL=0
MOVL C01794 V=800.0 PL=0
MOVL C01795 V=800.0 PL=0
MOVL C01796 V=800.0 PL=0
MOVL C01797 V=800.0 PL=0
MOVL C01798 V=800.0 PL=0
MOVL C01799 V=800.0 PL=0
MOVL C01800 V=800.0 PL=0
MOVL C01801 V=800.0 PL=0
MOVL C01802 V=800.0 PL=0
MOVL C01803 V=800.0 PL=0
MOVL C01804 V=800.0 PL=0
MOVL C01805 V=800.0 PL=0
MOVL C01806 V=800.0 PL=0
MOVL C01807 V=800.0 PL=0
MOVL C01808 V=800.0 PL=0
MOVL C01809 V=800.0 PL=0
MOVL C01810 V=800.0 PL=0
MOVL C01811 V=800.0 PL=0
MOVL C01812 V=800.0 PL=0
MOVL C01813 V=800.0 PL=0
MOVL C01814 V=800.0 PL=0
MOVL C01815 V=800.0 PL=0
MOVL C01816 V=800.0 PL=0
MOVL C01817 V=800.0 PL=0
MOVL C01818 V=800.0 PL=0
MOVL C01819 V=800.0 PL=0
MOVL C01820 V=800.0 PL=0
MOVL C01821 V=800.0 PL=0
MOVL C01822 V=800.0 PL=0
MOVL C01823 V=800.0 PL=0
MOVL C01824 V=800.0 PL=0
MOVL C01825 V=800.0 PL=0
MOVL C01826 V=800.0 PL=0
MOVL C01827 V=800.0 PL=0
MOVL C01828 V=800.0 PL=0
MOVL C01829 V=800.0 PL=0
MOVL C01830 V=800.0 PL=0
MOVL C01831 V=800.0 PL=0
MOVL C01832 V=800.0 PL=0
MOVL C01833 V=800.0 PL=0
MOVL C01834 V=800.0 PL=0
MOVL C01835 V=800.0 PL=0
MOVL C01836 V=800.0 PL=0
MOVL C01837 V=800.0 PL=0
MOVL C01838 V=800.0 PL=0
MOVL C01839 V=800.0 PL=0
MOVL C01840 V=800.0 PL=0
MOVL C01841 V=800.0 PL=0
MOVL C01842 V=800.0 PL=0
MOVL C01843 V=800.0 PL=0
MOVL C01844 V=800.0 PL=0
MOVL C01845 V=800.0 PL=0
MOVL C01846 V=800.0 PL=0
MOVL C01847 V=800.0 PL=0
MOVL C01848 V=800.0 PL=0
MOVL C01849 V=800.0 PL=0
MOVL C01850 V=800.0 PL=0
MOVL C01851 V=800.0 PL=0
MOVL C01852 V=800.0 PL=0
MOVL C01853 V=800.0 PL=0
MOVL C01854 V=800.0 PL=0
MOVL C01855 V=800.0 PL=0
MOVL C01856 V=800.0 PL=0
MOVL C01857 V=800.0 PL=0
MOVL C01858 V=800.0 PL=0
MOVL C01859 V=800.0 PL=0
MOVL C01860 V=800.0 PL=0
MOVL C01861 V=800.0 PL=0
MOVL C01862 V=800.0 PL=0
MOVL C01863 V=800.0 PL=0
MOVL C01864 V=800.0 PL=0
MOVL C01865 V=800.0 PL=0
MOVL C01866 V=800.0 PL=0
MOVL C01867 V=800.0 PL=0
MOVL C01868 V=800.0 PL=0
MOVL C01869 V=800.0 PL=0
MOVL C01870 V=800.0 PL=0
MOVL C01871 V=800.0 PL=0
MOVL C01872 V=800.0 PL=0
MOVL C01873 V=800.0 PL=0
MOVL C01874 V=800.0 PL=0
MOVL C01875 V=800.0 PL=0
MOVL C01876 V=800.0 PL=0
MOVL C01877 V=800.0 PL=0
MOVL C01878 V=800.0 PL=0
MOVL C01879 V=800.0 PL=0
MOVL C01880 V=800.0 PL=0
MOVL C01881 V=800.0 PL=0
MOVL C01882 V=800.0 PL=0
MOVL C01883 V=800.0 PL=0
MOVL C01884 V=800.0 PL=0
MOVL C01885 V=800.0 PL=0
MOVL C01886 V=800.0 PL=0
MOVL C01887 V=800.0 PL=0
MOVL C01888 V=800.0 PL=0
MOVL C01889 V=800.0 PL=0
MOVL C01890 V=800.0 PL=0
MOVL C01891 V=800.0 PL=0
MOVL C01892 V=800.0 PL=0
MOVL C01893 V=800.0 PL=0
MOVL C01894 V=800.0 PL=0
MOVL C01895 V=800.0 PL=0
MOVL C01896 V=800.0 PL=0
MOVL C01897 V=800.0 PL=0
MOVL C01898 V=800.0 PL=0
MOVL C01899 V=800.0 PL=0
MOVL C01900 V=800.0 PL=0
MOVL C01901 V=800.0 PL=0
MOVL C01902 V=800.0 PL=0
MOVL C01903 V=800.0 PL=0
MOVL C01904 V=800.0 PL=0
MOVL C01905 V=800.0 PL=0
MOVL C01906 V=800.0 PL=0
MOVL C01907 V=800.0 PL=0
MOVL C01908 V=800.0 PL=0
MOVL C01909 V=800.0 PL=0
MOVL C01910 V=800.0 PL=0
MOVL C01911 V=800.0 PL=0
MOVL C01912 V=800.0 PL=0
MOVL C01913 V=800.0 PL=0
MOVL C01914 V=800.0 PL=0
MOVL C01915 V=800.0 PL=0
MOVL C01916 V=800.0 PL=0
MOVL C01917 V=800.0 PL=0
MOVL C01918 V=800.0 PL=0
MOVL C01919 V=800.0 PL=0
MOVL C01920 V=800.0 PL=0
MOVL C01921 V=800.0 PL=0
